   LaserEnd_Ext()
   LIN {X -8.032, Y -15.360, Z 37.400}
   LaserStart_Ext()
   LIN {X 7.075, Y -15.360, Z 37.400}
   LaserEnd_Ext()
   LIN {X 7.240, Y -14.360, Z 37.400}
   LaserStart_Ext()
   LIN {X -7.569, Y -14.360, Z 37.400}
   LaserEnd_Ext()
   LIN {X -7.132, Y -13.360, Z 37.400}
   LaserStart_Ext()
   LIN {X 7.386, Y -13.360, Z 37.400}
   LaserEnd_Ext()
   LIN {X 7.511, Y -12.360, Z 37.400}
   LaserStart_Ext()
   LIN {X -6.697, Y -12.360, Z 37.400}
   LaserEnd_Ext()
   LIN {X -6.262, Y -11.360, Z 37.400}
   LaserStart_Ext()
   LIN {X 7.633, Y -11.360, Z 37.400}
   LaserEnd_Ext()
   LIN {X 7.756, Y -10.360, Z 37.400}
   LaserStart_Ext()
   LIN {X -5.884, Y -10.360, Z 37.400}
   LaserEnd_Ext()
   LIN {X -5.510, Y -9.360, Z 37.400}
   LaserStart_Ext()
   LIN {X 7.878, Y -9.360, Z 37.400}
   LaserEnd_Ext()
   LIN {X 7.959, Y -8.360, Z 37.400}
   LaserStart_Ext()
   LIN {X -5.135, Y -8.360, Z 37.400}
   LaserEnd_Ext()
   LIN {X -4.781, Y -7.360, Z 37.400}
   LaserStart_Ext()
   LIN {X 8.036, Y -7.360, Z 37.400}
   LaserEnd_Ext()
   LIN {X 8.113, Y -6.360, Z 37.400}
   LaserStart_Ext()
   LIN {X -4.476, Y -6.360, Z 37.400}
   LaserEnd_Ext()
   LIN {X -4.171, Y -5.360, Z 37.400}
   LaserStart_Ext()
   LIN {X 8.190, Y -5.360, Z 37.400}
   LaserEnd_Ext()
   LIN {X 8.267, Y -4.360, Z 37.400}
   LaserStart_Ext()
   LIN {X -3.865, Y -4.360, Z 37.400}
   LaserEnd_Ext()
   LIN {X -3.560, Y -3.360, Z 37.400}
   LaserStart_Ext()
   LIN {X 8.311, Y -3.360, Z 37.400}
   LaserEnd_Ext()
   LIN {X 8.326, Y -2.360, Z 37.400}
   LaserStart_Ext()
   LIN {X -3.286, Y -2.360, Z 37.400}
   LaserEnd_Ext()
   LIN {X -3.068, Y -1.360, Z 37.400}
   LaserStart_Ext()
   LIN {X 8.340, Y -1.360, Z 37.400}
   LaserEnd_Ext()
   LIN {X 8.355, Y -0.360, Z 37.400}
   LaserStart_Ext()
   LIN {X -2.851, Y -0.360, Z 37.400}
   LaserEnd_Ext()
   LIN {X -2.634, Y 0.640, Z 37.400}
   LaserStart_Ext()
   LIN {X 8.370, Y 0.640, Z 37.400}
   LaserEnd_Ext()
   LIN {X 8.384, Y 1.640, Z 37.400}
   LaserStart_Ext()
   LIN {X -2.417, Y 1.640, Z 37.400}
   LaserEnd_Ext()
   LIN {X -2.200, Y 2.640, Z 37.400}
   LaserStart_Ext()
   LIN {X 8.399, Y 2.640, Z 37.400}
   LaserEnd_Ext()
   LIN {X 8.413, Y 3.640, Z 37.400}
   LaserStart_Ext()
   LIN {X -1.983, Y 3.640, Z 37.400}
   LaserEnd_Ext()
   LIN {X -1.807, Y 4.640, Z 37.400}
   LaserStart_Ext()
   LIN {X 8.408, Y 4.640, Z 37.400}
   LaserEnd_Ext()
   LIN {X 8.352, Y 5.640, Z 37.400}
   LaserStart_Ext()
   LIN {X -1.698, Y 5.640, Z 37.400}
   LaserEnd_Ext()
   LIN {X -1.589, Y 6.640, Z 37.400}
   LaserStart_Ext()
   LIN {X 8.295, Y 6.640, Z 37.400}
   LaserEnd_Ext()
   LIN {X 8.239, Y 7.640, Z 37.400}
   LaserStart_Ext()
   LIN {X -1.481, Y 7.640, Z 37.400}
   LaserEnd_Ext()
   LIN {X -1.372, Y 8.640, Z 37.400}
   LaserStart_Ext()
   LIN {X 8.183, Y 8.640, Z 37.400}
   LaserEnd_Ext()
   LIN {X 8.135, Y 9.640, Z 37.400}
   LaserStart_Ext()
   LIN {X -1.263, Y 9.640, Z 37.400}
   LaserEnd_Ext()
   LIN {X -1.155, Y 10.640, Z 37.400}
   LaserStart_Ext()
   LIN {X 8.088, Y 10.640, Z 37.400}
   LaserEnd_Ext()
   LIN {X 8.007, Y 11.640, Z 37.400}
   LaserStart_Ext()
   LIN {X -1.046, Y 11.640, Z 37.400}
   LaserEnd_Ext()
   LIN {X -0.951, Y 12.640, Z 37.400}
   LaserStart_Ext()
   LIN {X 7.874, Y 12.640, Z 37.400}
   LaserEnd_Ext()
   LIN {X 7.735, Y 13.640, Z 37.400}
   LaserStart_Ext()
   LIN {X -0.969, Y 13.640, Z 37.400}
   LaserEnd_Ext()
   LIN {X -0.974, Y 14.640, Z 37.400}
   LaserStart_Ext()
   LIN {X 7.596, Y 14.640, Z 37.400}
   LaserEnd_Ext()
   LIN {X 7.457, Y 15.640, Z 37.400}
   LaserStart_Ext()
   LIN {X -0.979, Y 15.640, Z 37.400}
   LaserEnd_Ext()
   LIN {X -0.984, Y 16.640, Z 37.400}
   LaserStart_Ext()
   LIN {X 7.318, Y 16.640, Z 37.400}
   LaserEnd_Ext()
   LIN {X 7.179, Y 17.640, Z 37.400}
   LaserStart_Ext()
   LIN {X -0.990, Y 17.640, Z 37.400}
   LaserEnd_Ext()
   LIN {X -0.995, Y 18.640, Z 37.400}
   LaserStart_Ext()
   LIN {X 7.040, Y 18.640, Z 37.400}
   LaserEnd_Ext()
   LIN {X 6.901, Y 19.640, Z 37.400}
   LaserStart_Ext()
   LIN {X -1.000, Y 19.640, Z 37.400}
   LaserEnd_Ext()
   LIN {X -1.005, Y 20.640, Z 37.400}
   LaserStart_Ext()
   LIN {X 6.762, Y 20.640, Z 37.400}
   LaserEnd_Ext()
   LIN {X 6.617, Y 21.640, Z 37.400}
   LaserStart_Ext()
   LIN {X -1.081, Y 21.640, Z 37.400}
   LaserEnd_Ext()
   LIN {X -1.188, Y 22.640, Z 37.400}
   LaserStart_Ext()
   LIN {X 6.443, Y 22.640, Z 37.400}
   LaserEnd_Ext()
   LIN {X 6.225, Y 23.640, Z 37.400}
   LaserStart_Ext()
   LIN {X -1.295, Y 23.640, Z 37.400}
   LaserEnd_Ext()
   LIN {X -1.401, Y 24.640, Z 37.400}
   LaserStart_Ext()
   LIN {X 6.005, Y 24.640, Z 37.400}
   LaserEnd_Ext()
   LIN {X 5.784, Y 25.640, Z 37.400}
   LaserStart_Ext()
   LIN {X -1.508, Y 25.640, Z 37.400}
   LaserEnd_Ext()
   LIN {X -1.615, Y 26.640, Z 37.400}
   LaserStart_Ext()
   LIN {X 5.562, Y 26.640, Z 37.400}
   LaserEnd_Ext()
   LIN {X 5.340, Y 27.640, Z 37.400}
   LaserStart_Ext()
   LIN {X -1.725, Y 27.640, Z 37.400}
   LaserEnd_Ext()
   LIN {X -1.902, Y 28.640, Z 37.400}
   LaserStart_Ext()
   LIN {X 5.103, Y 28.640, Z 37.400}
   LaserEnd_Ext()
   LIN {X 4.836, Y 29.640, Z 37.400}
   LaserStart_Ext()
   LIN {X -2.078, Y 29.640, Z 37.400}
   LaserEnd_Ext()
   LIN {X -2.254, Y 30.640, Z 37.400}
   LaserStart_Ext()
   LIN {X 4.570, Y 30.640, Z 37.400}
   LaserEnd_Ext()
   LIN {X 4.298, Y 31.640, Z 37.400}
   LaserStart_Ext()
   LIN {X -2.465, Y 31.640, Z 37.400}
   LaserEnd_Ext()
   LIN {X -2.684, Y 32.640, Z 37.400}
   LaserStart_Ext()
   LIN {X 4.013, Y 32.640, Z 37.400}
   LaserEnd_Ext()
   LIN {X 3.709, Y 33.640, Z 37.400}
   LaserStart_Ext()
   LIN {X -2.905, Y 33.640, Z 37.400}
   LaserEnd_Ext()
   LIN {X -3.162, Y 34.640, Z 37.400}
   LaserStart_Ext()
   LIN {X 3.405, Y 34.640, Z 37.400}
   LaserEnd_Ext()
   LIN {X 3.089, Y 35.640, Z 37.400}
   LaserStart_Ext()
   LIN {X -3.420, Y 35.640, Z 37.400}
   LaserEnd_Ext()
   LIN {X -3.695, Y 36.640, Z 37.400}
   LaserStart_Ext()
   LIN {X 2.755, Y 36.640, Z 37.400}
   LaserEnd_Ext()
   LIN {X 2.422, Y 37.640, Z 37.400}
   LaserStart_Ext()
   LIN {X -3.984, Y 37.640, Z 37.400}
   LaserEnd_Ext()
   LIN {X -4.286, Y 38.640, Z 37.400}
   LaserStart_Ext()
   LIN {X 2.068, Y 38.640, Z 37.400}
   LaserEnd_Ext()
   LIN {X 1.708, Y 39.640, Z 37.400}
   LaserStart_Ext()
   LIN {X -4.427, Y 39.640, Z 37.400}
   LaserEnd_Ext()
   LIN {X -4.242, Y 40.640, Z 37.400}
   LaserStart_Ext()
   LIN {X 1.335, Y 40.640, Z 37.400}
   LaserEnd_Ext()
   LIN {X 0.726, Y 41.640, Z 37.400}
   LaserStart_Ext()
   LIN {X -3.673, Y 41.640, Z 37.400}
   LaserEnd_Ext()
   LIN {X -2.190, Y -26.841, Z 38.250}
   LaserStart_Ext()
   LIN {X -2.894, Y -26.717, Z 38.250} C_DIS
   LIN {X -4.205, Y -26.480, Z 38.250} C_DIS
   LIN {X -5.706, Y -25.455, Z 38.250} C_DIS
   LIN {X -5.911, Y -25.316, Z 38.250} C_DIS
   LIN {X -6.024, Y -25.134, Z 38.250} C_DIS
   LIN {X -7.009, Y -23.546, Z 38.250} C_DIS
   LIN {X -7.240, Y -21.756, Z 38.250} C_DIS
   LIN {X -7.277, Y -21.477, Z 38.250} C_DIS
   LIN {X -7.180, Y -21.203, Z 38.250} C_DIS
   LIN {X -6.319, Y -18.904, Z 38.250} C_DIS
   LIN {X -4.889, Y -17.604, Z 38.250} C_DIS
   LIN {X -4.667, Y -17.494, Z 38.250} C_DIS
   LIN {X -2.455, Y -16.842, Z 38.250} C_DIS
   LIN {X -1.080, Y -17.080, Z 38.250} C_DIS
   LIN {X -0.380, Y -17.198, Z 38.250} C_DIS
   LIN {X 0.350, Y -17.699, Z 38.250} C_DIS
   LIN {X 1.370, Y -18.402, Z 38.250} C_DIS
   LIN {X 2.014, Y -19.597, Z 38.250} C_DIS
   LIN {X 2.580, Y -20.639, Z 38.250} C_DIS
   LIN {X 2.596, Y -21.477, Z 38.250} C_DIS
   LIN {X 2.616, Y -22.815, Z 38.250} C_DIS
   LIN {X 2.128, Y -23.823, Z 38.250} C_DIS
   LIN {X 1.558, Y -25.016, Z 38.250} C_DIS
   LIN {X 0.417, Y -25.930, Z 38.250} C_DIS
   LIN {X -0.062, Y -26.310, Z 38.250} C_DIS
   LIN {X -1.069, Y -26.560, Z 38.250} C_DIS
   LIN {X -2.190, Y -26.841, Z 38.250}
   LaserEnd_Ext()
   LIN {X 3.341, Y 37.921, Z 38.250}
   LaserStart_Ext()
   LIN {X 2.785, Y 39.477, Z 38.250} C_DIS
   LIN {X 2.692, Y 39.739, Z 38.250} C_DIS
   LIN {X 2.643, Y 39.872, Z 38.250} C_DIS
   LIN {X 2.172, Y 41.130, Z 38.250} C_DIS
   LIN {X 1.504, Y 42.226, Z 38.250} C_DIS
   LIN {X 1.406, Y 42.387, Z 38.250} C_DIS
   LIN {X 1.194, Y 42.537, Z 38.250} C_DIS
   LIN {X -0.010, Y 43.401, Z 38.250} C_DIS
   LIN {X -1.088, Y 43.602, Z 38.250} C_DIS
   LIN {X -1.727, Y 43.719, Z 38.250} C_DIS
   LIN {X -3.855, Y 42.857, Z 38.250} C_DIS
   LIN {X -4.221, Y 42.712, Z 38.250} C_DIS
   LIN {X -5.222, Y 41.313, Z 38.250} C_DIS
   LIN {X -5.456, Y 40.383, Z 38.250} C_DIS
   LIN {X -5.540, Y 39.979, Z 38.250} C_DIS
   LIN {X -5.479, Y 39.534, Z 38.250} C_DIS
   LIN {X -5.349, Y 38.523, Z 38.250} C_DIS
   LIN {X -5.005, Y 37.398, Z 38.250} C_DIS
   LIN {X -4.937, Y 37.165, Z 38.250} C_DIS
   LIN {X -4.538, Y 35.789, Z 38.250} C_DIS
   LIN {X -4.133, Y 34.236, Z 38.250} C_DIS
   LIN {X -3.941, Y 33.495, Z 38.250} C_DIS
   LIN {X -3.664, Y 32.244, Z 38.250} C_DIS
   LIN {X -3.313, Y 30.668, Z 38.250} C_DIS
   LIN {X -3.137, Y 29.697, Z 38.250} C_DIS
   LIN {X -2.748, Y 27.508, Z 38.250} C_DIS
   LIN {X -2.473, Y 24.936, Z 38.250} C_DIS
   LIN {X -2.281, Y 23.139, Z 38.250} C_DIS
   LIN {X -2.204, Y 22.419, Z 38.250} C_DIS
   LIN {X -2.052, Y 21.233, Z 38.250} C_DIS
   LIN {X -2.015, Y 14.085, Z 38.250} C_DIS
   LIN {X -1.954, Y 12.608, Z 38.250} C_DIS
   LIN {X -2.361, Y 8.770, Z 38.250} C_DIS
   LIN {X -2.840, Y 4.366, Z 38.250} C_DIS
   LIN {X -3.751, Y 0.170, Z 38.250} C_DIS
   LIN {X -4.278, Y -2.326, Z 38.250} C_DIS
   LIN {X -4.552, Y -3.298, Z 38.250} C_DIS
   LIN {X -5.670, Y -6.961, Z 38.250} C_DIS
   LIN {X -6.324, Y -8.783, Z 38.250} C_DIS
   LIN {X -7.101, Y -10.858, Z 38.250} C_DIS
   LIN {X -8.557, Y -14.206, Z 38.250} C_DIS
   LIN {X -8.727, Y -14.604, Z 38.250} C_DIS
   LIN {X -8.883, Y -14.923, Z 38.250} C_DIS
   LIN {X -10.257, Y -17.683, Z 38.250} C_DIS
   LIN {X -11.156, Y -20.493, Z 38.250} C_DIS
   LIN {X -11.223, Y -20.704, Z 38.250} C_DIS
   LIN {X -11.210, Y -20.856, Z 38.250} C_DIS
   LIN {X -10.948, Y -24.404, Z 38.250} C_DIS
   LIN {X -9.577, Y -26.945, Z 38.250} C_DIS
   LIN {X -9.172, Y -27.706, Z 38.250} C_DIS
   LIN {X -8.750, Y -28.051, Z 38.250} C_DIS
   LIN {X -6.764, Y -29.691, Z 38.250} C_DIS
   LIN {X -3.576, Y -30.763, Z 38.250} C_DIS
   LIN {X -0.691, Y -30.694, Z 38.250} C_DIS
   LIN {X 2.555, Y -29.390, Z 38.250} C_DIS
   LIN {X 2.660, Y -29.342, Z 38.250} C_DIS
   LIN {X 2.800, Y -29.194, Z 38.250} C_DIS
   LIN {X 5.321, Y -26.624, Z 38.250} C_DIS
   LIN {X 5.995, Y -25.045, Z 38.250} C_DIS
   LIN {X 6.486, Y -23.872, Z 38.250} C_DIS
   LIN {X 7.011, Y -21.492, Z 38.250} C_DIS
   LIN {X 7.191, Y -20.687, Z 38.250} C_DIS
   LIN {X 7.275, Y -20.265, Z 38.250} C_DIS
   LIN {X 7.752, Y -17.779, Z 38.250} C_DIS
   LIN {X 8.260, Y -14.634, Z 38.250} C_DIS
   LIN {X 8.367, Y -13.948, Z 38.250} C_DIS
   LIN {X 8.494, Y -12.877, Z 38.250} C_DIS
   LIN {X 8.929, Y -9.318, Z 38.250} C_DIS
   LIN {X 9.169, Y -6.195, Z 38.250} C_DIS
   LIN {X 9.342, Y -3.768, Z 38.250} C_DIS
   LIN {X 9.340, Y -2.281, Z 38.250} C_DIS
   LIN {X 9.438, Y 4.467, Z 38.250} C_DIS
   LIN {X 9.114, Y 10.228, Z 38.250} C_DIS
   LIN {X 9.077, Y 11.017, Z 38.250} C_DIS
   LIN {X 9.049, Y 11.279, Z 38.250} C_DIS
   LIN {X 7.525, Y 22.243, Z 38.250} C_DIS
   LIN {X 7.508, Y 22.354, Z 38.250} C_DIS
   LIN {X 7.470, Y 22.528, Z 38.250} C_DIS
   LIN {X 6.118, Y 28.626, Z 38.250} C_DIS
   LIN {X 5.689, Y 30.237, Z 38.250} C_DIS
   LIN {X 5.004, Y 32.718, Z 38.250} C_DIS
   LIN {X 4.487, Y 34.418, Z 38.250} C_DIS
   LIN {X 3.908, Y 36.237, Z 38.250} C_DIS
   LIN {X 3.512, Y 37.422, Z 38.250} C_DIS
   LIN {X 3.341, Y 37.921, Z 38.250}
   LaserEnd_Ext()
   LIN {X 7.602, Y -11.930, Z 38.250}
   LaserStart_Ext()
   LIN {X 7.602, Y 14.428, Z 38.250}
   LaserEnd_Ext()
   LIN {X 6.602, Y 21.619, Z 38.250}
   LaserStart_Ext()
   LIN {X 6.602, Y -18.465, Z 38.250}
   LaserEnd_Ext()
   LIN {X 5.602, Y -23.239, Z 38.250}
   LaserStart_Ext()
   LIN {X 5.602, Y 26.334, Z 38.250}
   LaserEnd_Ext()
   LIN {X 4.602, Y 30.417, Z 38.250}
   LaserStart_Ext()
   LIN {X 4.602, Y -25.762, Z 38.250}
   LaserEnd_Ext()
   LIN {X 3.602, Y -26.949, Z 38.250}
   LaserStart_Ext()
   LIN {X 3.602, Y -22.979, Z 38.250}
   LaserEnd_Ext()
   LIN {X 3.602, Y -21.866, Z 38.250}
   LaserStart_Ext()
   LIN {X 3.602, Y 33.891, Z 38.250}
   LaserEnd_Ext()
   LIN {X 2.602, Y 36.989, Z 38.250}
   LaserStart_Ext()
   LIN {X 2.602, Y -18.581, Z 38.250}
   LaserEnd_Ext()
   LIN {X 2.602, Y -25.150, Z 38.250}
   LaserStart_Ext()
   LIN {X 2.602, Y -27.968, Z 38.250}
   LaserEnd_Ext()
   LIN {X 1.602, Y -28.696, Z 38.250}
   LaserStart_Ext()
   LIN {X 1.602, Y -26.262, Z 38.250}
   LaserEnd_Ext()
   LIN {X 1.602, Y -17.348, Z 38.250}
   LaserStart_Ext()
   LIN {X 1.602, Y 39.800, Z 38.250}
   LaserEnd_Ext()
   LIN {X 0.602, Y 41.732, Z 38.250}
   LaserStart_Ext()
   LIN {X 0.602, Y -16.659, Z 38.250}
   LaserEnd_Ext()
   LIN {X 0.602, Y -27.060, Z 38.250}
   LaserStart_Ext()
   LIN {X 0.602, Y -29.097, Z 38.250}
   LaserEnd_Ext()
   LIN {X -0.398, Y -29.499, Z 38.250}
   LaserStart_Ext()
   LIN {X -0.398, Y -27.424, Z 38.250}
   LaserEnd_Ext()
   LIN {X -0.398, Y -16.181, Z 38.250}
   LaserStart_Ext()
   LIN {X -0.398, Y 42.449, Z 38.250}
   LaserEnd_Ext()
   LIN {X -1.398, Y 42.642, Z 38.250}
   LaserStart_Ext()
   LIN {X -1.398, Y 24.288, Z 38.250}
   LaserEnd_Ext()
   LIN {X -1.398, Y 8.374, Z 38.250}
   LaserStart_Ext()
   LIN {X -1.398, Y -16.010, Z 38.250}
   LaserEnd_Ext()
   LIN {X -1.398, Y -27.674, Z 38.250}
   LaserStart_Ext()
   LIN {X -1.398, Y -29.713, Z 38.250}
   LaserEnd_Ext()
   LIN {X -2.398, Y -29.741, Z 38.250}
   LaserStart_Ext()
   LIN {X -2.398, Y -27.820, Z 38.250}
   LaserEnd_Ext()
   LIN {X -2.398, Y -15.845, Z 38.250}
   LaserStart_Ext()
   LIN {X -2.398, Y 1.687, Z 38.250}
   LaserEnd_Ext()
   LIN {X -2.398, Y 31.160, Z 38.250}
   LaserStart_Ext()
   LIN {X -2.398, Y 42.369, Z 38.250}
   LaserEnd_Ext()
   LIN {X -3.398, Y 41.964, Z 38.250}
   LaserStart_Ext()
   LIN {X -3.398, Y 35.380, Z 38.250}
   LaserEnd_Ext()
   LIN {X -3.398, Y -2.891, Z 38.250}
   LaserStart_Ext()
   LIN {X -3.398, Y -16.078, Z 38.250}
   LaserEnd_Ext()
   LIN {X -3.398, Y -27.642, Z 38.250}
   LaserStart_Ext()
   LIN {X -3.398, Y -29.768, Z 38.250}
   LaserEnd_Ext()
   LIN {X -4.398, Y -29.432, Z 38.250}
   LaserStart_Ext()
   LIN {X -4.398, Y -27.460, Z 38.250}
   LaserEnd_Ext()
   LIN {X -4.398, Y -16.372, Z 38.250}
   LaserStart_Ext()
   LIN {X -4.398, Y -6.218, Z 38.250}
   LaserEnd_Ext()
   LIN {X -4.398, Y 38.969, Z 38.250}
   LaserStart_Ext()
   LIN {X -4.398, Y 40.489, Z 38.250}
   LaserEnd_Ext()
   LIN {X -5.398, Y -9.162, Z 38.250}
   LaserStart_Ext()
   LIN {X -5.398, Y -16.724, Z 38.250}
   LaserEnd_Ext()
   LIN {X -5.398, Y -26.876, Z 38.250}
   LaserStart_Ext()
   LIN {X -5.398, Y -29.096, Z 38.250}
   LaserEnd_Ext()
   LIN {X -6.398, Y -28.696, Z 38.250}
   LaserStart_Ext()
   LIN {X -6.398, Y -26.194, Z 38.250}
   LaserEnd_Ext()
   LIN {X -6.398, Y -17.624, Z 38.250}
   LaserStart_Ext()
   LIN {X -6.398, Y -11.749, Z 38.250}
   LaserEnd_Ext()
   LIN {X -7.398, Y -14.049, Z 38.250}
   LaserStart_Ext()
   LIN {X -7.398, Y -18.934, Z 38.250}
   LaserEnd_Ext()
   LIN {X -7.398, Y -24.816, Z 38.250}
   LaserStart_Ext()
   LIN {X -7.398, Y -27.871, Z 38.250}
   LaserEnd_Ext()
   LIN {X -8.398, Y -27.033, Z 38.250}
   LaserStart_Ext()
   LIN {X -8.398, Y -16.192, Z 38.250}
   LaserEnd_Ext()
   LIN {X -9.398, Y -18.279, Z 38.250}
   LaserStart_Ext()
   LIN {X -9.398, Y -25.170, Z 38.250}
   LaserEnd_Ext()
   LIN {X -0.315, Y -17.145, Z 39.100}
   LaserStart_Ext()
   LIN {X 1.149, Y -18.149, Z 39.100} C_DIS
   LIN {X 1.438, Y -18.345, Z 39.100} C_DIS
   LIN {X 1.638, Y -18.710, Z 39.100} C_DIS
   LIN {X 2.654, Y -20.579, Z 39.100} C_DIS
   LIN {X 2.694, Y -22.707, Z 39.100} C_DIS
   LIN {X 1.640, Y -24.960, Z 39.100} C_DIS
   LIN {X 0.780, Y -25.649, Z 39.100} C_DIS
   LIN {X 0.024, Y -26.257, Z 39.100} C_DIS
   LIN {X -0.590, Y -26.413, Z 39.100} C_DIS
   LIN {X -2.102, Y -26.792, Z 39.100} C_DIS
   LIN {X -4.039, Y -26.450, Z 39.100} C_DIS
   LIN {X -4.208, Y -26.374, Z 39.100} C_DIS
   LIN {X -5.827, Y -25.276, Z 39.100} C_DIS
   LIN {X -6.722, Y -23.842, Z 39.100} C_DIS
   LIN {X -6.929, Y -23.508, Z 39.100} C_DIS
   LIN {X -6.977, Y -23.132, Z 39.100} C_DIS
   LIN {X -7.201, Y -21.440, Z 39.100} C_DIS
   LIN {X -6.612, Y -19.780, Z 39.100} C_DIS
   LIN {X -6.291, Y -18.921, Z 39.100} C_DIS
   LIN {X -5.757, Y -18.435, Z 39.100} C_DIS
   LIN {X -4.756, Y -17.498, Z 39.100} C_DIS
   LIN {X -2.486, Y -16.822, Z 39.100} C_DIS
   LIN {X -2.334, Y -16.804, Z 39.100} C_DIS
   LIN {X -0.315, Y -17.145, Z 39.100}
   LaserEnd_Ext()
   LIN {X 4.937, Y 32.834, Z 39.100}
   LaserStart_Ext()
   LIN {X 4.702, Y 33.610, Z 39.100} C_DIS
   LIN {X 3.734, Y 36.647, Z 39.100} C_DIS
   LIN {X 3.284, Y 37.964, Z 39.100} C_DIS
   LIN {X 3.129, Y 38.396, Z 39.100} C_DIS
   LIN {X 2.636, Y 39.768, Z 39.100} C_DIS
   LIN {X 2.116, Y 41.148, Z 39.100} C_DIS
   LIN {X 1.332, Y 42.444, Z 39.100} C_DIS
   LIN {X 0.139, Y 43.295, Z 39.100} C_DIS
   LIN {X -0.086, Y 43.454, Z 39.100} C_DIS
   LIN {X -0.617, Y 43.551, Z 39.100} C_DIS
   LIN {X -1.804, Y 43.769, Z 39.100} C_DIS
   LIN {X -2.601, Y 43.446, Z 39.100} C_DIS
   LIN {X -4.278, Y 42.771, Z 39.100} C_DIS
   LIN {X -5.066, Y 41.635, Z 39.100} C_DIS
   LIN {X -5.348, Y 41.235, Z 39.100} C_DIS
   LIN {X -5.411, Y 40.939, Z 39.100} C_DIS
   LIN {X -5.610, Y 39.982, Z 39.100} C_DIS
   LIN {X -5.450, Y 38.813, Z 39.100} C_DIS
   LIN {X -5.414, Y 38.564, Z 39.100} C_DIS
   LIN {X -5.356, Y 38.377, Z 39.100} C_DIS
   LIN {X -5.046, Y 37.368, Z 39.100} C_DIS
   LIN {X -4.693, Y 36.162, Z 39.100} C_DIS
   LIN {X -4.597, Y 35.833, Z 39.100} C_DIS
   LIN {X -4.434, Y 35.207, Z 39.100} C_DIS
   LIN {X -3.994, Y 33.539, Z 39.100} C_DIS
   LIN {X -3.673, Y 32.120, Z 39.100} C_DIS
   LIN {X -3.359, Y 30.714, Z 39.100} C_DIS
   LIN {X -2.838, Y 27.832, Z 39.100} C_DIS
   LIN {X -2.787, Y 27.556, Z 39.100} C_DIS
   LIN {X -2.482, Y 24.705, Z 39.100} C_DIS
   LIN {X -2.353, Y 23.493, Z 39.100} C_DIS
   LIN {X -2.097, Y 21.497, Z 39.100} C_DIS
   LIN {X -2.064, Y 15.178, Z 39.100} C_DIS
   LIN {X -1.959, Y 12.611, Z 39.100} C_DIS
   LIN {X -2.666, Y 5.940, Z 39.100} C_DIS
   LIN {X -2.843, Y 4.309, Z 39.100} C_DIS
   LIN {X -3.180, Y 2.756, Z 39.100} C_DIS
   LIN {X -4.227, Y -2.202, Z 39.100} C_DIS
   LIN {X -4.772, Y -4.132, Z 39.100} C_DIS
   LIN {X -5.541, Y -6.652, Z 39.100} C_DIS
   LIN {X -6.740, Y -9.994, Z 39.100} C_DIS
   LIN {X -7.039, Y -10.793, Z 39.100} C_DIS
   LIN {X -7.599, Y -12.080, Z 39.100} C_DIS
   LIN {X -8.627, Y -14.480, Z 39.100} C_DIS
   LIN {X -9.566, Y -16.399, Z 39.100} C_DIS
   LIN {X -10.191, Y -17.653, Z 39.100} C_DIS
   LIN {X -10.599, Y -18.930, Z 39.100} C_DIS
   LIN {X -11.149, Y -20.676, Z 39.100} C_DIS
   LIN {X -11.046, Y -21.940, Z 39.100} C_DIS
   LIN {X -10.865, Y -24.376, Z 39.100} C_DIS
   LIN {X -9.367, Y -27.154, Z 39.100} C_DIS
   LIN {X -9.082, Y -27.674, Z 39.100} C_DIS
   LIN {X -8.700, Y -27.993, Z 39.100} C_DIS
   LIN {X -6.732, Y -29.617, Z 39.100} C_DIS
   LIN {X -4.570, Y -30.344, Z 39.100} C_DIS
   LIN {X -3.417, Y -30.730, Z 39.100} C_DIS
   LIN {X -2.188, Y -30.662, Z 39.100} C_DIS
   LIN {X -0.453, Y -30.614, Z 39.100} C_DIS
   LIN {X 1.494, Y -29.832, Z 39.100} C_DIS
   LIN {X 2.883, Y -29.187, Z 39.100} C_DIS
   LIN {X 4.742, Y -27.235, Z 39.100} C_DIS
   LIN {X 5.413, Y -26.552, Z 39.100} C_DIS
   LIN {X 5.592, Y -26.132, Z 39.100} C_DIS
   LIN {X 6.568, Y -23.803, Z 39.100} C_DIS
   LIN {X 7.099, Y -21.392, Z 39.100} C_DIS
   LIN {X 7.265, Y -20.616, Z 39.100} C_DIS
   LIN {X 7.478, Y -19.484, Z 39.100} C_DIS
   LIN {X 7.819, Y -17.707, Z 39.100} C_DIS
   LIN {X 8.077, Y -16.110, Z 39.100} C_DIS
   LIN {X 8.423, Y -13.892, Z 39.100} C_DIS
   LIN {X 8.831, Y -10.433, Z 39.100} C_DIS
   LIN {X 8.974, Y -9.261, Z 39.100} C_DIS
   LIN {X 9.053, Y -8.233, Z 39.100} C_DIS
   LIN {X 9.376, Y -3.680, Z 39.100} C_DIS
   LIN {X 9.374, Y -0.891, Z 39.100} C_DIS
   LIN {X 9.453, Y 4.552, Z 39.100} C_DIS
   LIN {X 9.129, Y 10.300, Z 39.100} C_DIS
   LIN {X 9.051, Y 11.219, Z 39.100} C_DIS
   LIN {X 8.866, Y 12.442, Z 39.100} C_DIS
   LIN {X 7.477, Y 22.438, Z 39.100} C_DIS
   LIN {X 6.434, Y 27.075, Z 39.100} C_DIS
   LIN {X 6.067, Y 28.732, Z 39.100} C_DIS
   LIN {X 5.962, Y 29.123, Z 39.100} C_DIS
   LIN {X 4.937, Y 32.834, Z 39.100}
   LaserEnd_Ext()
   LIN {X -0.546, Y 42.522, Z 39.100}
   LaserStart_Ext()
   LIN {X -2.219, Y 42.522, Z 39.100}
   LaserEnd_Ext()
   LIN {X -3.928, Y 41.522, Z 39.100}
   LaserStart_Ext()
   LIN {X 0.724, Y 41.522, Z 39.100}
   LaserEnd_Ext()
   LIN {X 1.283, Y 40.522, Z 39.100}
   LaserStart_Ext()
   LIN {X -4.476, Y 40.522, Z 39.100}
   LaserEnd_Ext()
   LIN {X -4.538, Y 39.522, Z 39.100}
   LaserStart_Ext()
   LIN {X 1.660, Y 39.522, Z 39.100}
   LaserEnd_Ext()
   LIN {X 2.021, Y 38.522, Z 39.100}
   LaserStart_Ext()
   LIN {X -4.354, Y 38.522, Z 39.100}
   LaserEnd_Ext()
   LIN {X -4.049, Y 37.522, Z 39.100}
   LaserStart_Ext()
   LIN {X 2.378, Y 37.522, Z 39.100}
   LaserEnd_Ext()
   LIN {X 2.721, Y 36.522, Z 39.100}
   LaserStart_Ext()
   LIN {X -3.756, Y 36.522, Z 39.100}
   LaserEnd_Ext()
   LIN {X -3.482, Y 35.522, Z 39.100}
   LaserStart_Ext()
   LIN {X 3.043, Y 35.522, Z 39.100}
   LaserEnd_Ext()
   LIN {X 3.362, Y 34.522, Z 39.100}
   LaserStart_Ext()
   LIN {X -3.219, Y 34.522, Z 39.100}
   LaserEnd_Ext()
   LIN {X -2.965, Y 33.522, Z 39.100}
   LaserStart_Ext()
   LIN {X 3.680, Y 33.522, Z 39.100}
   LaserEnd_Ext()
   LIN {X 3.986, Y 32.522, Z 39.100}
   LaserStart_Ext()
   LIN {X -2.739, Y 32.522, Z 39.100}
   LaserEnd_Ext()
   LIN {X -2.515, Y 31.522, Z 39.100}
   LaserStart_Ext()
   LIN {X 4.262, Y 31.522, Z 39.100}
   LaserEnd_Ext()
   LIN {X 4.539, Y 30.522, Z 39.100}
   LaserStart_Ext()
   LIN {X -2.308, Y 30.522, Z 39.100}
   LaserEnd_Ext()
   LIN {X -2.127, Y 29.522, Z 39.100}
   LaserStart_Ext()
   LIN {X 4.815, Y 29.522, Z 39.100}
   LaserEnd_Ext()
   LIN {X 5.088, Y 28.522, Z 39.100}
   LaserStart_Ext()
   LIN {X -1.946, Y 28.522, Z 39.100}
   LaserEnd_Ext()
   LIN {X -1.778, Y 27.522, Z 39.100}
   LaserStart_Ext()
   LIN {X 5.311, Y 27.522, Z 39.100}
   LaserEnd_Ext()
   LIN {X 5.534, Y 26.522, Z 39.100}
   LaserStart_Ext()
   LIN {X -1.671, Y 26.522, Z 39.100}
   LaserEnd_Ext()
   LIN {X -1.564, Y 25.522, Z 39.100}
   LaserStart_Ext()
   LIN {X 5.759, Y 25.522, Z 39.100}
   LaserEnd_Ext()
   LIN {X 5.984, Y 24.522, Z 39.100}
   LaserStart_Ext()
   LIN {X -1.457, Y 24.522, Z 39.100}
   LaserEnd_Ext()
   LIN {X -1.348, Y 23.522, Z 39.100}
   LaserStart_Ext()
   LIN {X 6.209, Y 23.522, Z 39.100}
   LaserEnd_Ext()
   LIN {X 6.434, Y 22.522, Z 39.100}
   LaserStart_Ext()
   LIN {X -1.220, Y 22.522, Z 39.100}
   LaserEnd_Ext()
   LIN {X -1.099, Y 21.522, Z 39.100}
   LaserStart_Ext()
   LIN {X 6.595, Y 21.522, Z 39.100}
   LaserEnd_Ext()
   LIN {X 6.734, Y 20.522, Z 39.100}
   LaserStart_Ext()
   LIN {X -1.092, Y 20.522, Z 39.100}
   LaserEnd_Ext()
   LIN {X -1.087, Y 19.522, Z 39.100}
   LaserStart_Ext()
   LIN {X 6.873, Y 19.522, Z 39.100}
   LaserEnd_Ext()
   LIN {X 7.012, Y 18.522, Z 39.100}
   LaserStart_Ext()
   LIN {X -1.082, Y 18.522, Z 39.100}
   LaserEnd_Ext()
   LIN {X -1.076, Y 17.522, Z 39.100}
   LaserStart_Ext()
   LIN {X 7.151, Y 17.522, Z 39.100}
   LaserEnd_Ext()
   LIN {X 7.290, Y 16.522, Z 39.100}
   LaserStart_Ext()
   LIN {X -1.071, Y 16.522, Z 39.100}
   LaserEnd_Ext()
   LIN {X -1.066, Y 15.522, Z 39.100}
   LaserStart_Ext()
   LIN {X 7.429, Y 15.522, Z 39.100}
   LaserEnd_Ext()
   LIN {X 7.568, Y 14.522, Z 39.100}
   LaserStart_Ext()
   LIN {X -1.037, Y 14.522, Z 39.100}
   LaserEnd_Ext()
   LIN {X -0.996, Y 13.522, Z 39.100}
   LaserStart_Ext()
   LIN {X 7.707, Y 13.522, Z 39.100}
   LaserEnd_Ext()
   LIN {X 7.846, Y 12.522, Z 39.100}
   LaserStart_Ext()
   LIN {X -0.964, Y 12.522, Z 39.100}
   LaserEnd_Ext()
   LIN {X -1.069, Y 11.522, Z 39.100}
   LaserStart_Ext()
   LIN {X 7.994, Y 11.522, Z 39.100}
   LaserEnd_Ext()
   LIN {X 8.107, Y 10.522, Z 39.100}
   LaserStart_Ext()
   LIN {X -1.175, Y 10.522, Z 39.100}
   LaserEnd_Ext()
   LIN {X -1.281, Y 9.522, Z 39.100}
   LaserStart_Ext()
   LIN {X 8.171, Y 9.522, Z 39.100}
   LaserEnd_Ext()
   LIN {X 8.228, Y 8.522, Z 39.100}
   LaserStart_Ext()
   LIN {X -1.387, Y 8.522, Z 39.100}
   LaserEnd_Ext()
   LIN {X -1.493, Y 7.522, Z 39.100}
   LaserStart_Ext()
   LIN {X 8.284, Y 7.522, Z 39.100}
   LaserEnd_Ext()
   LIN {X 8.340, Y 6.522, Z 39.100}
   LaserStart_Ext()
   LIN {X -1.599, Y 6.522, Z 39.100}
   LaserEnd_Ext()
   LIN {X -1.705, Y 5.522, Z 39.100}
   LaserStart_Ext()
   LIN {X 8.396, Y 5.522, Z 39.100}
   LaserEnd_Ext()
   LIN {X 8.452, Y 4.522, Z 39.100}
   LaserStart_Ext()
   LIN {X -1.814, Y 4.522, Z 39.100}
   LaserEnd_Ext()
   LIN {X -1.991, Y 3.522, Z 39.100}
   LaserStart_Ext()
   LIN {X 8.438, Y 3.522, Z 39.100}
   LaserEnd_Ext()
   LIN {X 8.423, Y 2.522, Z 39.100}
   LaserStart_Ext()
   LIN {X -2.208, Y 2.522, Z 39.100}
   LaserEnd_Ext()
   LIN {X -2.419, Y 1.522, Z 39.100}
   LaserStart_Ext()
   LIN {X 8.409, Y 1.522, Z 39.100}
   LaserEnd_Ext()
   LIN {X 8.394, Y 0.522, Z 39.100}
   LaserStart_Ext()
   LIN {X -2.630, Y 0.522, Z 39.100}
   LaserEnd_Ext()
   LIN {X -2.841, Y -0.478, Z 39.100}
   LaserStart_Ext()
   LIN {X 8.379, Y -0.478, Z 39.100}
   LaserEnd_Ext()
   LIN {X 8.374, Y -1.478, Z 39.100}
   LaserStart_Ext()
   LIN {X -3.052, Y -1.478, Z 39.100}
   LaserEnd_Ext()
   LIN {X -3.266, Y -2.478, Z 39.100}
   LaserStart_Ext()
   LIN {X 8.375, Y -2.478, Z 39.100}
   LaserEnd_Ext()
   LIN {X 8.376, Y -3.478, Z 39.100}
   LaserStart_Ext()
   LIN {X -3.548, Y -3.478, Z 39.100}
   LaserEnd_Ext()
   LIN {X -3.832, Y -4.478, Z 39.100}
   LaserStart_Ext()
   LIN {X 8.317, Y -4.478, Z 39.100}
   LaserEnd_Ext()
   LIN {X 8.246, Y -5.478, Z 39.100}
   LaserStart_Ext()
   LIN {X -4.137, Y -5.478, Z 39.100}
   LaserEnd_Ext()
   LIN {X -4.443, Y -6.478, Z 39.100}
   LaserStart_Ext()
   LIN {X 8.175, Y -6.478, Z 39.100}
   LaserEnd_Ext()
   LIN {X 8.104, Y -7.478, Z 39.100}
   LaserStart_Ext()
   LIN {X -4.775, Y -7.478, Z 39.100}
   LaserEnd_Ext()
   LIN {X -5.134, Y -8.478, Z 39.100}
   LaserStart_Ext()
   LIN {X 8.031, Y -8.478, Z 39.100}
   LaserEnd_Ext()
   LIN {X 7.940, Y -9.478, Z 39.100}
   LaserStart_Ext()
   LIN {X -5.493, Y -9.478, Z 39.100}
   LaserEnd_Ext()
   LIN {X -5.854, Y -10.478, Z 39.100}
   LaserStart_Ext()
   LIN {X 7.818, Y -10.478, Z 39.100}
   LaserEnd_Ext()
   LIN {X 7.700, Y -11.478, Z 39.100}
   LaserStart_Ext()
   LIN {X -6.247, Y -11.478, Z 39.100}
   LaserEnd_Ext()
   LIN {X -6.682, Y -12.478, Z 39.100}
   LaserStart_Ext()
   LIN {X 7.583, Y -12.478, Z 39.100}
   LaserEnd_Ext()
   LIN {X 7.465, Y -13.478, Z 39.100}
   LaserStart_Ext()
   LIN {X -7.110, Y -13.478, Z 39.100}
   LaserEnd_Ext()
   LIN {X -7.538, Y -14.478, Z 39.100}
   LaserStart_Ext()
   LIN {X 7.319, Y -14.478, Z 39.100}
   LaserEnd_Ext()
   LIN {X 7.163, Y -15.478, Z 39.100}
   LaserStart_Ext()
   LIN {X -8.002, Y -15.478, Z 39.100}
   LaserEnd_Ext()
   LIN {X -8.492, Y -16.478, Z 39.100}
   LaserStart_Ext()
   LIN {X -4.836, Y -16.478, Z 39.100}
   LaserEnd_Ext()
   LIN {X 0.481, Y -16.478, Z 39.100}
   LaserStart_Ext()
   LIN {X 7.004, Y -16.478, Z 39.100}
   LaserEnd_Ext()
   LIN {X 6.843, Y -17.478, Z 39.100}
   LaserStart_Ext()
   LIN {X 1.942, Y -17.478, Z 39.100}
   LaserEnd_Ext()
   LIN {X -6.198, Y -17.478, Z 39.100}
   LaserStart_Ext()
   LIN {X -8.987, Y -17.478, Z 39.100}
   LaserEnd_Ext()
   LIN {X -9.405, Y -18.478, Z 39.100}
   LaserStart_Ext()
   LIN {X -7.187, Y -18.478, Z 39.100}
   LaserEnd_Ext()
   LIN {X 2.650, Y -18.478, Z 39.100}
   LaserStart_Ext()
   LIN {X 6.652, Y -18.478, Z 39.100}
   LaserEnd_Ext()
   LIN {X 6.461, Y -19.478, Z 39.100}
   LaserStart_Ext()
   LIN {X 3.194, Y -19.478, Z 39.100}
   LaserEnd_Ext()
   LIN {X -7.567, Y -19.478, Z 39.100}
   LaserStart_Ext()
   LIN {X -9.724, Y -19.478, Z 39.100}
   LaserEnd_Ext()
   LIN {X -10.038, Y -20.478, Z 39.100}
   LaserStart_Ext()
   LIN {X -7.921, Y -20.478, Z 39.100}
   LaserEnd_Ext()
   LIN {X 3.648, Y -20.478, Z 39.100}
   LaserStart_Ext()
   LIN {X 6.272, Y -20.478, Z 39.100}
   LaserEnd_Ext()
   LIN {X 6.056, Y -21.478, Z 39.100}
   LaserStart_Ext()
   LIN {X 3.671, Y -21.478, Z 39.100}
   LaserEnd_Ext()
   LIN {X -8.201, Y -21.478, Z 39.100}
   LaserStart_Ext()
   LIN {X -10.080, Y -21.478, Z 39.100}
   LaserEnd_Ext()
   LIN {X -10.003, Y -22.478, Z 39.100}
   LaserStart_Ext()
   LIN {X -8.073, Y -22.478, Z 39.100}
   LaserEnd_Ext()
   LIN {X 3.690, Y -22.478, Z 39.100}
   LaserStart_Ext()
   LIN {X 5.836, Y -22.478, Z 39.100}
   LaserEnd_Ext()
   LIN {X 5.615, Y -23.478, Z 39.100}
   LaserStart_Ext()
   LIN {X 3.457, Y -23.478, Z 39.100}
   LaserEnd_Ext()
   LIN {X -7.941, Y -23.478, Z 39.100}
   LaserStart_Ext()
   LIN {X -9.929, Y -23.478, Z 39.100}
   LaserEnd_Ext()
   LIN {X -9.674, Y -24.478, Z 39.100}
   LaserStart_Ext()
   LIN {X -7.504, Y -24.478, Z 39.100}
   LaserEnd_Ext()
   LIN {X 2.979, Y -24.478, Z 39.100}
   LaserStart_Ext()
   LIN {X 5.201, Y -24.478, Z 39.100}
   LaserEnd_Ext()
   LIN {X 4.782, Y -25.478, Z 39.100}
   LaserStart_Ext()
   LIN {X 2.495, Y -25.478, Z 39.100}
   LaserEnd_Ext()
   LIN {X -6.879, Y -25.478, Z 39.100}
   LaserStart_Ext()
   LIN {X -9.134, Y -25.478, Z 39.100}
   LaserEnd_Ext()
   LIN {X -8.595, Y -26.478, Z 39.100}
   LaserStart_Ext()
   LIN {X -5.835, Y -26.478, Z 39.100}
   LaserEnd_Ext()
   LIN {X 1.344, Y -26.478, Z 39.100}
   LaserStart_Ext()
   LIN {X 4.084, Y -26.478, Z 39.100}
   LaserEnd_Ext()
   LIN {X 3.130, Y -27.478, Z 39.100}
   LaserStart_Ext()
   LIN {X -0.726, Y -27.478, Z 39.100}
   LaserEnd_Ext()
   LIN {X -3.966, Y -27.478, Z 39.100}
   LaserStart_Ext()
   LIN {X -7.752, Y -27.478, Z 39.100}
   LaserEnd_Ext()
   LIN {X -6.541, Y -28.478, Z 39.100}
   LaserStart_Ext()
   LIN {X 2.035, Y -28.478, Z 39.100}
   LaserEnd_Ext()
   LIN {X -0.308, Y -29.478, Z 39.100}
   LaserStart_Ext()
   LIN {X -4.007, Y -29.478, Z 39.100}
   LaserEnd_Ext()
   LIN {X -4.691, Y -17.456, Z 39.950}
   LaserStart_Ext()
   LIN {X -3.638, Y -17.142, Z 39.950} C_DIS
   LIN {X -2.328, Y -16.746, Z 39.950} C_DIS
   LIN {X -0.755, Y -17.006, Z 39.950} C_DIS
   LIN {X -0.250, Y -17.092, Z 39.950} C_DIS
   LIN {X 0.094, Y -17.327, Z 39.950} C_DIS
   LIN {X 1.506, Y -18.288, Z 39.950} C_DIS
   LIN {X 2.484, Y -20.071, Z 39.950} C_DIS
   LIN {X 2.728, Y -20.518, Z 39.950} C_DIS
   LIN {X 2.738, Y -21.055, Z 39.950} C_DIS
   LIN {X 2.773, Y -22.694, Z 39.950} C_DIS
   LIN {X 1.923, Y -24.477, Z 39.950} C_DIS
   LIN {X 1.732, Y -24.892, Z 39.950} C_DIS
   LIN {X 1.292, Y -25.253, Z 39.950} C_DIS
   LIN {X 0.111, Y -26.203, Z 39.950} C_DIS
   LIN {X -1.760, Y -26.680, Z 39.950} C_DIS
   LIN {X -2.014, Y -26.743, Z 39.950} C_DIS
   LIN {X -2.372, Y -26.680, Z 39.950} C_DIS
   LIN {X -4.030, Y -26.391, Z 39.950} C_DIS
   LIN {X -5.098, Y -25.672, Z 39.950} C_DIS
   LIN {X -5.742, Y -25.235, Z 39.950} C_DIS
   LIN {X -6.222, Y -24.467, Z 39.950} C_DIS
   LIN {X -6.848, Y -23.471, Z 39.950} C_DIS
   LIN {X -7.013, Y -22.255, Z 39.950} C_DIS
   LIN {X -7.126, Y -21.403, Z 39.950} C_DIS
   LIN {X -6.632, Y -20.009, Z 39.950} C_DIS
   LIN {X -6.232, Y -18.895, Z 39.950} C_DIS
   LIN {X -5.712, Y -18.412, Z 39.950} C_DIS
   LIN {X -4.691, Y -17.456, Z 39.950}
   LaserEnd_Ext()
   LIN {X -2.142, Y 21.760, Z 39.950}
   LaserStart_Ext()
   LIN {X -2.502, Y 24.567, Z 39.950} C_DIS
   LIN {X -2.684, Y 26.271, Z 39.950} C_DIS
   LIN {X -2.826, Y 27.603, Z 39.950} C_DIS
   LIN {X -3.244, Y 29.885, Z 39.950} C_DIS
   LIN {X -3.406, Y 30.760, Z 39.950} C_DIS
   LIN {X -3.696, Y 32.032, Z 39.950} C_DIS
   LIN {X -4.047, Y 33.584, Z 39.950} C_DIS
   LIN {X -4.261, Y 34.395, Z 39.950} C_DIS
   LIN {X -4.655, Y 35.875, Z 39.950} C_DIS
   LIN {X -5.094, Y 37.364, Z 39.950} C_DIS
   LIN {X -5.479, Y 38.605, Z 39.950} C_DIS
   LIN {X -5.650, Y 39.786, Z 39.950} C_DIS
   LIN {X -5.679, Y 39.997, Z 39.950} C_DIS
   LIN {X -5.622, Y 40.258, Z 39.950} C_DIS
   LIN {X -5.396, Y 41.334, Z 39.950} C_DIS
   LIN {X -4.720, Y 42.292, Z 39.950} C_DIS
   LIN {X -4.330, Y 42.836, Z 39.950} C_DIS
   LIN {X -3.909, Y 43.003, Z 39.950} C_DIS
   LIN {X -1.882, Y 43.818, Z 39.950} C_DIS
   LIN {X -1.118, Y 43.682, Z 39.950} C_DIS
   LIN {X -0.163, Y 43.508, Z 39.950} C_DIS
   LIN {X 1.235, Y 42.516, Z 39.950} C_DIS
   LIN {X 2.030, Y 41.247, Z 39.950} C_DIS
   LIN {X 2.488, Y 40.039, Z 39.950} C_DIS
   LIN {X 2.581, Y 39.792, Z 39.950} C_DIS
   LIN {X 2.731, Y 39.377, Z 39.950} C_DIS
   LIN {X 3.267, Y 37.893, Z 39.950} C_DIS
   LIN {X 3.554, Y 37.055, Z 39.950} C_DIS
   LIN {X 3.936, Y 35.912, Z 39.950} C_DIS
   LIN {X 4.856, Y 32.997, Z 39.950} C_DIS
   LIN {X 4.920, Y 32.781, Z 39.950} C_DIS
   LIN {X 6.015, Y 28.838, Z 39.950} C_DIS
   LIN {X 6.322, Y 27.525, Z 39.950} C_DIS
   LIN {X 7.442, Y 22.548, Z 39.950} C_DIS
   LIN {X 8.442, Y 15.351, Z 39.950} C_DIS
   LIN {X 8.989, Y 11.729, Z 39.950} C_DIS
   LIN {X 9.221, Y 9.006, Z 39.950} C_DIS
   LIN {X 9.467, Y 4.636, Z 39.950} C_DIS
   LIN {X 9.407, Y 0.499, Z 39.950} C_DIS
   LIN {X 9.410, Y -3.593, Z 39.950} C_DIS
   LIN {X 9.110, Y -7.828, Z 39.950} C_DIS
   LIN {X 9.020, Y -9.189, Z 39.950} C_DIS
   LIN {X 8.919, Y -10.097, Z 39.950} C_DIS
   LIN {X 8.478, Y -13.836, Z 39.950} C_DIS
   LIN {X 7.893, Y -17.586, Z 39.950} C_DIS
   LIN {X 7.875, Y -17.689, Z 39.950} C_DIS
   LIN {X 7.339, Y -20.544, Z 39.950} C_DIS
   LIN {X 6.920, Y -22.504, Z 39.950} C_DIS
   LIN {X 6.649, Y -23.734, Z 39.950} C_DIS
   LIN {X 5.935, Y -25.437, Z 39.950} C_DIS
   LIN {X 5.504, Y -26.479, Z 39.950} C_DIS
   LIN {X 5.032, Y -27.011, Z 39.950} C_DIS
   LIN {X 3.105, Y -29.032, Z 39.950} C_DIS
   LIN {X 0.434, Y -30.273, Z 39.950} C_DIS
   LIN {X -0.214, Y -30.534, Z 39.950} C_DIS
   LIN {X -0.792, Y -30.550, Z 39.950} C_DIS
   LIN {X -3.284, Y -30.688, Z 39.950} C_DIS
   LIN {X -5.623, Y -29.906, Z 39.950} C_DIS
   LIN {X -6.701, Y -29.543, Z 39.950} C_DIS
   LIN {X -7.682, Y -28.733, Z 39.950} C_DIS
   LIN {X -8.992, Y -27.641, Z 39.950} C_DIS
   LIN {X -9.969, Y -25.857, Z 39.950} C_DIS
   LIN {X -10.783, Y -24.347, Z 39.950} C_DIS
   LIN {X -10.881, Y -23.024, Z 39.950} C_DIS
   LIN {X -11.075, Y -20.648, Z 39.950} C_DIS
   LIN {X -10.173, Y -17.782, Z 39.950} C_DIS
   LIN {X -10.124, Y -17.624, Z 39.950} C_DIS
   LIN {X -10.002, Y -17.369, Z 39.950} C_DIS
   LIN {X -8.527, Y -14.356, Z 39.950} C_DIS
   LIN {X -7.199, Y -11.257, Z 39.950} C_DIS
   LIN {X -6.978, Y -10.727, Z 39.950} C_DIS
   LIN {X -6.587, Y -9.618, Z 39.950} C_DIS
   LIN {X -5.412, Y -6.343, Z 39.950} C_DIS
   LIN {X -4.992, Y -4.966, Z 39.950} C_DIS
   LIN {X -4.177, Y -2.077, Z 39.950} C_DIS
   LIN {X -2.937, Y 3.795, Z 39.950} C_DIS
   LIN {X -2.841, Y 4.282, Z 39.950} C_DIS
   LIN {X -2.823, Y 4.501, Z 39.950} C_DIS
   LIN {X -1.964, Y 12.614, Z 39.950} C_DIS
   LIN {X -2.114, Y 16.272, Z 39.950} C_DIS
   LIN {X -2.142, Y 21.760, Z 39.950}
   LaserEnd_Ext()
   LIN {X -9.280, Y -25.028, Z 39.950}
   LaserStart_Ext()
   LIN {X -9.280, Y -18.275, Z 39.950}
   LaserEnd_Ext()
   LIN {X -8.280, Y -16.126, Z 39.950}
   LaserStart_Ext()
   LIN {X -8.280, Y -26.859, Z 39.950}
   LaserEnd_Ext()
   LIN {X -7.280, Y -27.767, Z 39.950}
   LaserStart_Ext()
   LIN {X -7.280, Y -24.663, Z 39.950}
   LaserEnd_Ext()
   LIN {X -7.280, Y -18.855, Z 39.950}
   LaserStart_Ext()
   LIN {X -7.280, Y -13.985, Z 39.950}
   LaserEnd_Ext()
   LIN {X -6.280, Y -11.650, Z 39.950}
   LaserStart_Ext()
   LIN {X -6.280, Y -17.574, Z 39.950}
   LaserEnd_Ext()
   LIN {X -6.280, Y -26.079, Z 39.950}
   LaserStart_Ext()
   LIN {X -6.280, Y -28.594, Z 39.950}
   LaserEnd_Ext()
   LIN {X -5.280, Y -28.966, Z 39.950}
   LaserStart_Ext()
   LIN {X -5.280, Y -26.755, Z 39.950}
   LaserEnd_Ext()
   LIN {X -5.280, Y -16.649, Z 39.950}
   LaserStart_Ext()
   LIN {X -5.280, Y -8.935, Z 39.950}
   LaserEnd_Ext()
   LIN {X -4.280, Y 41.181, Z 39.950}
   LaserStart_Ext()
   LIN {X -4.280, Y 38.116, Z 39.950}
   LaserEnd_Ext()
   LIN {X -4.280, Y -6.058, Z 39.950}
   LaserStart_Ext()
   LIN {X -4.280, Y -16.290, Z 39.950}
   LaserEnd_Ext()
   LIN {X -4.280, Y -27.359, Z 39.950}
   LaserStart_Ext()
   LIN {X -4.280, Y -29.301, Z 39.950}
   LaserEnd_Ext()
   LIN {X -3.280, Y -29.635, Z 39.950}
   LaserStart_Ext()
   LIN {X -3.280, Y -27.537, Z 39.950}
   LaserEnd_Ext()
   LIN {X -3.280, Y -15.989, Z 39.950}
   LaserStart_Ext()
   LIN {X -3.280, Y -2.581, Z 39.950}
   LaserEnd_Ext()
   LIN {X -3.280, Y 34.596, Z 39.950}
   LaserStart_Ext()
   LIN {X -3.280, Y 42.178, Z 39.950}
   LaserEnd_Ext()
   LIN {X -2.280, Y 42.580, Z 39.950}
   LaserStart_Ext()
   LIN {X -2.280, Y 30.172, Z 39.950}
   LaserEnd_Ext()
   LIN {X -2.280, Y 2.065, Z 39.950}
   LaserStart_Ext()
   LIN {X -2.280, Y -15.748, Z 39.950}
   LaserEnd_Ext()
   LIN {X -2.280, Y -27.712, Z 39.950}
   LaserStart_Ext()
   LIN {X -2.280, Y -29.631, Z 39.950}
   LaserEnd_Ext()
   LIN {X -1.280, Y -29.575, Z 39.950}
   LaserStart_Ext()
   LIN {X -1.280, Y -27.589, Z 39.950}
   LaserEnd_Ext()
   LIN {X -1.280, Y -15.906, Z 39.950}
   LaserStart_Ext()
   LIN {X -1.280, Y 9.578, Z 39.950}
   LaserEnd_Ext()
   LIN {X -1.280, Y 22.898, Z 39.950}
   LaserStart_Ext()
   LIN {X -1.280, Y 42.695, Z 39.950}
   LaserEnd_Ext()
   LIN {X -0.280, Y 42.365, Z 39.950}
   LaserStart_Ext()
   LIN {X -0.280, Y -16.072, Z 39.950}
   LaserEnd_Ext()
   LIN {X -0.280, Y -27.334, Z 39.950}
   LaserStart_Ext()
   LIN {X -0.280, Y -29.482, Z 39.950}
   LaserEnd_Ext()
   LIN {X 0.720, Y -29.038, Z 39.950}
   LaserStart_Ext()
   LIN {X 0.720, Y -26.995, Z 39.950}
   LaserEnd_Ext()
   LIN {X 0.720, Y -16.544, Z 39.950}
   LaserStart_Ext()
   LIN {X 0.720, Y 41.466, Z 39.950}
   LaserEnd_Ext()
   LIN {X 1.720, Y 39.231, Z 39.950}
   LaserStart_Ext()
   LIN {X 1.720, Y -17.224, Z 39.950}
   LaserEnd_Ext()
   LIN {X 1.720, Y -26.192, Z 39.950}
   LaserStart_Ext()
   LIN {X 1.720, Y -28.573, Z 39.950}
   LaserEnd_Ext()
   LIN {X 2.720, Y -27.987, Z 39.950}
   LaserStart_Ext()
   LIN {X 2.720, Y -25.137, Z 39.950}
   LaserEnd_Ext()
   LIN {X 2.720, Y -18.421, Z 39.950}
   LaserStart_Ext()
   LIN {X 2.720, Y 36.396, Z 39.950}
   LaserEnd_Ext()
   LIN {X 3.720, Y 33.274, Z 39.950}
   LaserStart_Ext()
   LIN {X 3.720, Y -20.398, Z 39.950}
   LaserEnd_Ext()
   LIN {X 3.720, Y -23.013, Z 39.950}
   LaserStart_Ext()
   LIN {X 3.720, Y -26.938, Z 39.950}
   LaserEnd_Ext()
   LIN {X 4.720, Y -25.759, Z 39.950}
   LaserStart_Ext()
   LIN {X 4.720, Y 29.763, Z 39.950}
   LaserEnd_Ext()
   LIN {X 5.720, Y 25.646, Z 39.950}
   LaserStart_Ext()
   LIN {X 5.720, Y -23.301, Z 39.950}
   LaserEnd_Ext()
   LIN {X 6.720, Y -18.421, Z 39.950}
   LaserStart_Ext()
   LIN {X 6.720, Y 20.480, Z 39.950}
   LaserEnd_Ext()
   LIN {X 7.720, Y 13.435, Z 39.950}
   LaserStart_Ext()
   LIN {X 7.720, Y -11.725, Z 39.950}
   LaserEnd_Ext()
   LIN {X 2.196, Y -19.364, Z 40.800}
   LaserStart_Ext()
   LIN {X 2.801, Y -20.458, Z 40.800} C_DIS
   LIN {X 2.826, Y -21.415, Z 40.800} C_DIS
   LIN {X 2.852, Y -22.634, Z 40.800} C_DIS
   LIN {X 2.456, Y -23.464, Z 40.800} C_DIS
   LIN {X 1.835, Y -24.810, Z 40.800} C_DIS
   LIN {X 0.409, Y -25.979, Z 40.800} C_DIS
   LIN {X 0.198, Y -26.149, Z 40.800} C_DIS
   LIN {X -0.258, Y -26.265, Z 40.800} C_DIS
   LIN {X -1.926, Y -26.694, Z 40.800} C_DIS
   LIN {X -2.951, Y -26.519, Z 40.800} C_DIS
   LIN {X -3.943, Y -26.347, Z 40.800} C_DIS
   LIN {X -5.040, Y -25.608, Z 40.800} C_DIS
   LIN {X -5.657, Y -25.195, Z 40.800} C_DIS
   LIN {X -6.000, Y -24.654, Z 40.800} C_DIS
   LIN {X -6.768, Y -23.433, Z 40.800} C_DIS
   LIN {X -6.955, Y -22.051, Z 40.800} C_DIS
   LIN {X -7.050, Y -21.365, Z 40.800} C_DIS
   LIN {X -6.781, Y -20.631, Z 40.800} C_DIS
   LIN {X -6.126, Y -18.806, Z 40.800} C_DIS
   LIN {X -4.853, Y -17.623, Z 40.800} C_DIS
   LIN {X -4.595, Y -17.396, Z 40.800} C_DIS
   LIN {X -4.162, Y -17.272, Z 40.800} C_DIS
   LIN {X -2.263, Y -16.697, Z 40.800} C_DIS
   LIN {X -1.062, Y -16.896, Z 40.800} C_DIS
   LIN {X -0.184, Y -17.038, Z 40.800} C_DIS
   LIN {X 0.687, Y -17.626, Z 40.800} C_DIS
   LIN {X 1.575, Y -18.230, Z 40.800} C_DIS
   LIN {X 2.196, Y -19.364, Z 40.800}
   LaserEnd_Ext()
   LIN {X 8.214, Y -15.831, Z 40.800}
   LaserStart_Ext()
   LIN {X 7.952, Y -17.562, Z 40.800} C_DIS
   LIN {X 7.735, Y -18.754, Z 40.800} C_DIS
   LIN {X 7.413, Y -20.473, Z 40.800} C_DIS
   LIN {X 6.741, Y -23.616, Z 40.800} C_DIS
   LIN {X 6.702, Y -23.730, Z 40.800} C_DIS
   LIN {X 5.596, Y -26.406, Z 40.800} C_DIS
   LIN {X 4.381, Y -27.773, Z 40.800} C_DIS
   LIN {X 3.328, Y -28.878, Z 40.800} C_DIS
   LIN {X 0.988, Y -29.965, Z 40.800} C_DIS
   LIN {X 0.023, Y -30.447, Z 40.800} C_DIS
   LIN {X -0.770, Y -30.514, Z 40.800} C_DIS
   LIN {X -3.152, Y -30.646, Z 40.800} C_DIS
   LIN {X -6.656, Y -29.474, Z 40.800} C_DIS
   LIN {X -8.902, Y -27.608, Z 40.800} C_DIS
   LIN {X -10.570, Y -24.560, Z 40.800} C_DIS
   LIN {X -10.701, Y -24.319, Z 40.800} C_DIS
   LIN {X -10.716, Y -24.107, Z 40.800} C_DIS
   LIN {X -11.001, Y -20.620, Z 40.800} C_DIS
   LIN {X -10.398, Y -18.703, Z 40.800} C_DIS
   LIN {X -10.057, Y -17.593, Z 40.800} C_DIS
   LIN {X -9.202, Y -15.816, Z 40.800} C_DIS
   LIN {X -8.426, Y -14.233, Z 40.800} C_DIS
   LIN {X -7.729, Y -12.604, Z 40.800} C_DIS
   LIN {X -6.916, Y -10.661, Z 40.800} C_DIS
   LIN {X -5.484, Y -6.593, Z 40.800} C_DIS
   LIN {X -5.283, Y -6.034, Z 40.800} C_DIS
   LIN {X -5.212, Y -5.799, Z 40.800} C_DIS
   LIN {X -4.126, Y -1.953, Z 40.800} C_DIS
   LIN {X -3.159, Y 2.626, Z 40.800} C_DIS
   LIN {X -2.830, Y 4.297, Z 40.800} C_DIS
   LIN {X -2.771, Y 5.046, Z 40.800} C_DIS
   LIN {X -1.969, Y 12.617, Z 40.800} C_DIS
   LIN {X -2.163, Y 17.365, Z 40.800} C_DIS
   LIN {X -2.187, Y 22.023, Z 40.800} C_DIS
   LIN {X -2.651, Y 25.641, Z 40.800} C_DIS
   LIN {X -2.865, Y 27.650, Z 40.800} C_DIS
   LIN {X -2.966, Y 28.185, Z 40.800} C_DIS
   LIN {X -3.452, Y 30.805, Z 40.800} C_DIS
   LIN {X -3.778, Y 32.234, Z 40.800} C_DIS
   LIN {X -4.100, Y 33.628, Z 40.800} C_DIS
   LIN {X -4.494, Y 35.093, Z 40.800} C_DIS
   LIN {X -4.714, Y 35.918, Z 40.800} C_DIS
   LIN {X -4.829, Y 36.307, Z 40.800} C_DIS
   LIN {X -5.170, Y 37.452, Z 40.800} C_DIS
   LIN {X -5.475, Y 38.428, Z 40.800} C_DIS
   LIN {X -5.544, Y 38.646, Z 40.800} C_DIS
   LIN {X -5.599, Y 39.056, Z 40.800} C_DIS
   LIN {X -5.744, Y 40.100, Z 40.800} C_DIS
   LIN {X -5.573, Y 40.881, Z 40.800} C_DIS
   LIN {X -5.425, Y 41.471, Z 40.800} C_DIS
   LIN {X -4.797, Y 42.321, Z 40.800} C_DIS
   LIN {X -4.381, Y 42.900, Z 40.800} C_DIS
   LIN {X -2.603, Y 43.608, Z 40.800} C_DIS
   LIN {X -1.959, Y 43.867, Z 40.800} C_DIS
   LIN {X -0.892, Y 43.677, Z 40.800} C_DIS
   LIN {X -0.239, Y 43.561, Z 40.800} C_DIS
   LIN {X 0.096, Y 43.325, Z 40.800} C_DIS
   LIN {X 1.184, Y 42.557, Z 40.800} C_DIS
   LIN {X 1.871, Y 41.447, Z 40.800} C_DIS
   LIN {X 1.959, Y 41.305, Z 40.800} C_DIS
   LIN {X 2.035, Y 41.104, Z 40.800} C_DIS
   LIN {X 2.506, Y 39.873, Z 40.800} C_DIS
   LIN {X 2.960, Y 38.625, Z 40.800} C_DIS
   LIN {X 3.265, Y 37.780, Z 40.800} C_DIS
   LIN {X 3.374, Y 37.462, Z 40.800} C_DIS
   LIN {X 4.162, Y 35.106, Z 40.800} C_DIS
   LIN {X 4.697, Y 33.411, Z 40.800} C_DIS
   LIN {X 5.157, Y 31.846, Z 40.800} C_DIS
   LIN {X 5.963, Y 28.943, Z 40.800} C_DIS
   LIN {X 6.723, Y 25.698, Z 40.800} C_DIS
   LIN {X 7.407, Y 22.657, Z 40.800} C_DIS
   LIN {X 8.018, Y 18.260, Z 40.800} C_DIS
   LIN {X 8.927, Y 12.238, Z 40.800} C_DIS
   LIN {X 9.313, Y 7.712, Z 40.800} C_DIS
   LIN {X 9.481, Y 4.721, Z 40.800} C_DIS
   LIN {X 9.440, Y 1.889, Z 40.800} C_DIS
   LIN {X 9.445, Y -3.505, Z 40.800} C_DIS
   LIN {X 9.334, Y -5.070, Z 40.800} C_DIS
   LIN {X 9.068, Y -9.102, Z 40.800} C_DIS
   LIN {X 8.768, Y -11.791, Z 40.800} C_DIS
   LIN {X 8.534, Y -13.780, Z 40.800} C_DIS
   LIN {X 8.214, Y -15.831, Z 40.800}
   LaserEnd_Ext()
   LIN {X -3.844, Y -29.360, Z 40.800}
   LaserStart_Ext()
   LIN {X -0.039, Y -29.360, Z 40.800}
   LaserEnd_Ext()
   LIN {X 2.069, Y -28.360, Z 40.800}
   LaserStart_Ext()
   LIN {X -6.438, Y -28.360, Z 40.800}
   LaserEnd_Ext()
   LIN {X -7.638, Y -27.360, Z 40.800}
   LaserStart_Ext()
   LIN {X -3.952, Y -27.360, Z 40.800}
   LaserEnd_Ext()
   LIN {X -0.502, Y -27.360, Z 40.800}
   LaserStart_Ext()
   LIN {X 3.393, Y -27.360, Z 40.800}
   LaserEnd_Ext()
   LIN {X 4.299, Y -26.360, Z 40.800}
   LaserStart_Ext()
   LIN {X 1.521, Y -26.360, Z 40.800}
   LaserEnd_Ext()
   LIN {X -5.714, Y -26.360, Z 40.800}
   LaserStart_Ext()
   LIN {X -8.445, Y -26.360, Z 40.800}
   LaserEnd_Ext()
   LIN {X -8.993, Y -25.360, Z 40.800}
   LaserStart_Ext()
   LIN {X -6.737, Y -25.360, Z 40.800}
   LaserEnd_Ext()
   LIN {X 2.669, Y -25.360, Z 40.800}
   LaserStart_Ext()
   LIN {X 4.946, Y -25.360, Z 40.800}
   LaserEnd_Ext()
   LIN {X 5.360, Y -24.360, Z 40.800}
   LaserStart_Ext()
   LIN {X 3.144, Y -24.360, Z 40.800}
   LaserEnd_Ext()
   LIN {X -7.366, Y -24.360, Z 40.800}
   LaserStart_Ext()
   LIN {X -9.540, Y -24.360, Z 40.800}
   LaserEnd_Ext()
   LIN {X -9.774, Y -23.360, Z 40.800}
   LaserStart_Ext()
   LIN {X -7.787, Y -23.360, Z 40.800}
   LaserEnd_Ext()
   LIN {X 3.613, Y -23.360, Z 40.800}
   LaserStart_Ext()
   LIN {X 5.773, Y -23.360, Z 40.800}
   LaserEnd_Ext()
   LIN {X 5.987, Y -22.360, Z 40.800}
   LaserStart_Ext()
   LIN {X 3.846, Y -22.360, Z 40.800}
   LaserEnd_Ext()
   LIN {X -7.922, Y -22.360, Z 40.800}
   LaserStart_Ext()
   LIN {X -9.856, Y -22.360, Z 40.800}
   LaserEnd_Ext()
   LIN {X -9.938, Y -21.360, Z 40.800}
   LaserStart_Ext()
   LIN {X -8.049, Y -21.360, Z 40.800}
   LaserEnd_Ext()
   LIN {X 3.825, Y -21.360, Z 40.800}
   LaserStart_Ext()
   LIN {X 6.200, Y -21.360, Z 40.800}
   LaserEnd_Ext()
   LIN {X 6.414, Y -20.360, Z 40.800}
   LaserStart_Ext()
   LIN {X 3.796, Y -20.360, Z 40.800}
   LaserEnd_Ext()
   LIN {X -7.747, Y -20.360, Z 40.800}
   LaserStart_Ext()
   LIN {X -9.871, Y -20.360, Z 40.800}
   LaserEnd_Ext()
   LIN {X -9.556, Y -19.360, Z 40.800}
   LaserStart_Ext()
   LIN {X -7.388, Y -19.360, Z 40.800}
   LaserEnd_Ext()
   LIN {X 3.337, Y -19.360, Z 40.800}
   LaserStart_Ext()
   LIN {X 6.604, Y -19.360, Z 40.800}
   LaserEnd_Ext()
   LIN {X 6.791, Y -18.360, Z 40.800}
   LaserStart_Ext()
   LIN {X 2.787, Y -18.360, Z 40.800}
   LaserEnd_Ext()
   LIN {X -7.020, Y -18.360, Z 40.800}
   LaserStart_Ext()
   LIN {X -9.247, Y -18.360, Z 40.800}
   LaserEnd_Ext()
   LIN {X -8.835, Y -17.360, Z 40.800}
   LaserStart_Ext()
   LIN {X -6.039, Y -17.360, Z 40.800}
   LaserEnd_Ext()
   LIN {X 2.074, Y -17.360, Z 40.800}
   LaserStart_Ext()
   LIN {X 6.972, Y -17.360, Z 40.800}
   LaserEnd_Ext()
   LIN {X 7.123, Y -16.360, Z 40.800}
   LaserStart_Ext()
   LIN {X 0.599, Y -16.360, Z 40.800}
   LaserEnd_Ext()
   LIN {X -4.609, Y -16.360, Z 40.800}
   LaserStart_Ext()
   LIN {X -8.354, Y -16.360, Z 40.800}
   LaserEnd_Ext()
   LIN {X -7.865, Y -15.360, Z 40.800}
   LaserStart_Ext()
   LIN {X 7.275, Y -15.360, Z 40.800}
   LaserEnd_Ext()
   LIN {X 7.431, Y -14.360, Z 40.800}
   LaserStart_Ext()
   LIN {X -7.393, Y -14.360, Z 40.800}
   LaserEnd_Ext()
   LIN {X -6.965, Y -13.360, Z 40.800}
   LaserStart_Ext()
   LIN {X 7.576, Y -13.360, Z 40.800}
   LaserEnd_Ext()
   LIN {X 7.694, Y -12.360, Z 40.800}
   LaserStart_Ext()
   LIN {X -6.543, Y -12.360, Z 40.800}
   LaserEnd_Ext()
   LIN {X -6.125, Y -11.360, Z 40.800}
   LaserStart_Ext()
   LIN {X 7.810, Y -11.360, Z 40.800}
   LaserEnd_Ext()
   LIN {X 7.922, Y -10.360, Z 40.800}
   LaserStart_Ext()
   LIN {X -5.750, Y -10.360, Z 40.800}
   LaserEnd_Ext()
   LIN {X -5.398, Y -9.360, Z 40.800}
   LaserStart_Ext()
   LIN {X 8.033, Y -9.360, Z 40.800}
   LaserEnd_Ext()
   LIN {X 8.115, Y -8.360, Z 40.800}
   LaserStart_Ext()
   LIN {X -5.046, Y -8.360, Z 40.800}
   LaserEnd_Ext()
   LIN {X -4.694, Y -7.360, Z 40.800}
   LaserStart_Ext()
   LIN {X 8.181, Y -7.360, Z 40.800}
   LaserEnd_Ext()
   LIN {X 8.247, Y -6.360, Z 40.800}
   LaserStart_Ext()
   LIN {X -4.338, Y -6.360, Z 40.800}
   LaserEnd_Ext()
   LIN {X -4.049, Y -5.360, Z 40.800}
   LaserStart_Ext()
   LIN {X 8.313, Y -5.360, Z 40.800}
   LaserEnd_Ext()
   LIN {X 8.382, Y -4.360, Z 40.800}
   LaserStart_Ext()
   LIN {X -3.766, Y -4.360, Z 40.800}
   LaserEnd_Ext()
   LIN {X -3.484, Y -3.360, Z 40.800}
   LaserStart_Ext()
   LIN {X 8.445, Y -3.360, Z 40.800}
   LaserEnd_Ext()
   LIN {X 8.444, Y -2.360, Z 40.800}
   LaserStart_Ext()
   LIN {X -3.202, Y -2.360, Z 40.800}
   LaserEnd_Ext()
   LIN {X -2.979, Y -1.360, Z 40.800}
   LaserStart_Ext()
   LIN {X 8.443, Y -1.360, Z 40.800}
   LaserEnd_Ext()
   LIN {X 8.442, Y -0.360, Z 40.800}
   LaserStart_Ext()
   LIN {X -2.768, Y -0.360, Z 40.800}
   LaserEnd_Ext()
   LIN {X -2.557, Y 0.640, Z 40.800}
   LaserStart_Ext()
   LIN {X 8.441, Y 0.640, Z 40.800}
   LaserEnd_Ext()
   LIN {X 8.440, Y 1.640, Z 40.800}
   LaserStart_Ext()
   LIN {X -2.345, Y 1.640, Z 40.800}
   LaserEnd_Ext()
   LIN {X -2.137, Y 2.640, Z 40.800}
   LaserStart_Ext()
   LIN {X 8.451, Y 2.640, Z 40.800}
   LaserEnd_Ext()
   LIN {X 8.465, Y 3.640, Z 40.800}
   LaserStart_Ext()
   LIN {X -1.940, Y 3.640, Z 40.800}
   LaserEnd_Ext()
   LIN {X -1.800, Y 4.640, Z 40.800}
   LaserStart_Ext()
   LIN {X 8.480, Y 4.640, Z 40.800}
   LaserEnd_Ext()
   LIN {X 8.428, Y 5.640, Z 40.800}
   LaserStart_Ext()
   LIN {X -1.702, Y 5.640, Z 40.800}
   LaserEnd_Ext()
   LIN {X -1.596, Y 6.640, Z 40.800}
   LaserStart_Ext()
   LIN {X 8.372, Y 6.640, Z 40.800}
   LaserEnd_Ext()
   LIN {X 8.315, Y 7.640, Z 40.800}
   LaserStart_Ext()
   LIN {X -1.490, Y 7.640, Z 40.800}
   LaserEnd_Ext()
   LIN {X -1.384, Y 8.640, Z 40.800}
   LaserStart_Ext()
   LIN {X 8.230, Y 8.640, Z 40.800}
   LaserEnd_Ext()
   LIN {X 8.145, Y 9.640, Z 40.800}
   LaserStart_Ext()
   LIN {X -1.278, Y 9.640, Z 40.800}
   LaserEnd_Ext()
   LIN {X -1.172, Y 10.640, Z 40.800}
   LaserStart_Ext()
   LIN {X 8.060, Y 10.640, Z 40.800}
   LaserEnd_Ext()
   LIN {X 7.975, Y 11.640, Z 40.800}
   LaserStart_Ext()
   LIN {X -1.067, Y 11.640, Z 40.800}
   LaserEnd_Ext()
   LIN {X -0.970, Y 12.640, Z 40.800}
   LaserStart_Ext()
   LIN {X 7.855, Y 12.640, Z 40.800}
   LaserEnd_Ext()
   LIN {X 7.704, Y 13.640, Z 40.800}
   LaserStart_Ext()
   LIN {X -1.010, Y 13.640, Z 40.800}
   LaserEnd_Ext()
   LIN {X -1.051, Y 14.640, Z 40.800}
   LaserStart_Ext()
   LIN {X 7.553, Y 14.640, Z 40.800}
   LaserEnd_Ext()
   LIN {X 7.402, Y 15.640, Z 40.800}
   LaserStart_Ext()
   LIN {X -1.092, Y 15.640, Z 40.800}
   LaserEnd_Ext()
   LIN {X -1.133, Y 16.640, Z 40.800}
   LaserStart_Ext()
   LIN {X 7.252, Y 16.640, Z 40.800}
   LaserEnd_Ext()
   LIN {X 7.101, Y 17.640, Z 40.800}
   LaserStart_Ext()
   LIN {X -1.165, Y 17.640, Z 40.800}
   LaserEnd_Ext()
   LIN {X -1.170, Y 18.640, Z 40.800}
   LaserStart_Ext()
   LIN {X 6.956, Y 18.640, Z 40.800}
   LaserEnd_Ext()
   LIN {X 6.817, Y 19.640, Z 40.800}
   LaserStart_Ext()
   LIN {X -1.175, Y 19.640, Z 40.800}
   LaserEnd_Ext()
   LIN {X -1.180, Y 20.640, Z 40.800}
   LaserStart_Ext()
   LIN {X 6.678, Y 20.640, Z 40.800}
   LaserEnd_Ext()
   LIN {X 6.539, Y 21.640, Z 40.800}
   LaserStart_Ext()
   LIN {X -1.185, Y 21.640, Z 40.800}
   LaserEnd_Ext()
   LIN {X -1.258, Y 22.640, Z 40.800}
   LaserStart_Ext()
   LIN {X 6.386, Y 22.640, Z 40.800}
   LaserEnd_Ext()
   LIN {X 6.161, Y 23.640, Z 40.800}
   LaserStart_Ext()
   LIN {X -1.386, Y 23.640, Z 40.800}
   LaserEnd_Ext()
   LIN {X -1.514, Y 24.640, Z 40.800}
   LaserStart_Ext()
   LIN {X 5.936, Y 24.640, Z 40.800}
   LaserEnd_Ext()
   LIN {X 5.710, Y 25.640, Z 40.800}
   LaserStart_Ext()
   LIN {X -1.642, Y 25.640, Z 40.800}
   LaserEnd_Ext()
   LIN {X -1.752, Y 26.640, Z 40.800}
   LaserStart_Ext()
   LIN {X 5.475, Y 26.640, Z 40.800}
   LaserEnd_Ext()
   LIN {X 5.241, Y 27.640, Z 40.800}
   LaserStart_Ext()
   LIN {X -1.859, Y 27.640, Z 40.800}
   LaserEnd_Ext()
   LIN {X -2.033, Y 28.640, Z 40.800}
   LaserStart_Ext()
   LIN {X 5.007, Y 28.640, Z 40.800}
   LaserEnd_Ext()
   LIN {X 4.731, Y 29.640, Z 40.800}
   LaserStart_Ext()
   LIN {X -2.219, Y 29.640, Z 40.800}
   LaserEnd_Ext()
   LIN {X -2.405, Y 30.640, Z 40.800}
   LaserStart_Ext()
   LIN {X 4.454, Y 30.640, Z 40.800}
   LaserEnd_Ext()
   LIN {X 4.175, Y 31.640, Z 40.800}
   LaserStart_Ext()
   LIN {X -2.617, Y 31.640, Z 40.800}
   LaserEnd_Ext()
   LIN {X -2.846, Y 32.640, Z 40.800}
   LaserStart_Ext()
   LIN {X 3.881, Y 32.640, Z 40.800}
   LaserEnd_Ext()
   LIN {X 3.576, Y 33.640, Z 40.800}
   LaserStart_Ext()
   LIN {X -3.077, Y 33.640, Z 40.800}
   LaserEnd_Ext()
   LIN {X -3.337, Y 34.640, Z 40.800}
   LaserStart_Ext()
   LIN {X 3.260, Y 34.640, Z 40.800}
   LaserEnd_Ext()
   LIN {X 2.929, Y 35.640, Z 40.800}
   LaserStart_Ext()
   LIN {X -3.605, Y 35.640, Z 40.800}
   LaserEnd_Ext()
   LIN {X -3.884, Y 36.640, Z 40.800}
   LaserStart_Ext()
   LIN {X 2.594, Y 36.640, Z 40.800}
   LaserEnd_Ext()
   LIN {X 2.252, Y 37.640, Z 40.800}
   LaserStart_Ext()
   LIN {X -4.182, Y 37.640, Z 40.800}
   LaserEnd_Ext()
   LIN {X -4.494, Y 38.640, Z 40.800}
   LaserStart_Ext()
   LIN {X 1.890, Y 38.640, Z 40.800}
   LaserEnd_Ext()
   LIN {X 1.524, Y 39.640, Z 40.800}
   LaserStart_Ext()
   LIN {X -4.671, Y 39.640, Z 40.800}
   LaserEnd_Ext()
   LIN {X -4.602, Y 40.640, Z 40.800}
   LaserStart_Ext()
   LIN {X 1.142, Y 40.640, Z 40.800}
   LaserEnd_Ext()
   LIN {X 0.575, Y 41.640, Z 40.800}
   LaserStart_Ext()
   LIN {X -4.056, Y 41.640, Z 40.800}
   LaserEnd_Ext()
   LIN {X -2.331, Y 42.640, Z 40.800}
   LaserStart_Ext()
   LIN {X -0.773, Y 42.640, Z 40.800}
   LaserEnd_Ext()
   LIN {X -6.975, Y -21.328, Z 41.650}
   LaserStart_Ext()
   LIN {X -6.151, Y -19.080, Z 41.650} C_DIS
   LIN {X -6.021, Y -18.717, Z 41.650} C_DIS
   LIN {X -5.767, Y -18.481, Z 41.650} C_DIS
   LIN {X -4.394, Y -17.279, Z 41.650} C_DIS
   LIN {X -2.259, Y -16.665, Z 41.650} C_DIS
   LIN {X -2.116, Y -16.662, Z 41.650} C_DIS
   LIN {X -0.118, Y -16.985, Z 41.650} C_DIS
   LIN {X 1.314, Y -17.952, Z 41.650} C_DIS
   LIN {X 1.643, Y -18.173, Z 41.650} C_DIS
   LIN {X 1.894, Y -18.622, Z 41.650} C_DIS
   LIN {X 2.875, Y -20.397, Z 41.650} C_DIS
   LIN {X 2.925, Y -22.355, Z 41.650} C_DIS
   LIN {X 2.931, Y -22.573, Z 41.650} C_DIS
   LIN {X 2.661, Y -23.163, Z 41.650} C_DIS
   LIN {X 1.939, Y -24.727, Z 41.650} C_DIS
   LIN {X 1.443, Y -25.133, Z 41.650} C_DIS
   LIN {X 0.271, Y -26.101, Z 41.650} C_DIS
   LIN {X -1.837, Y -26.644, Z 41.650} C_DIS
   LIN {X -3.453, Y -26.370, Z 41.650} C_DIS
   LIN {X -3.855, Y -26.302, Z 41.650} C_DIS
   LIN {X -4.115, Y -26.130, Z 41.650} C_DIS
   LIN {X -5.573, Y -25.154, Z 41.650} C_DIS
   LIN {X -6.668, Y -23.426, Z 41.650} C_DIS
   LIN {X -6.975, Y -21.328, Z 41.650}
   LaserEnd_Ext()
   LIN {X -4.365, Y 34.461, Z 41.650}
   LaserStart_Ext()
   LIN {X -4.772, Y 35.961, Z 41.650} C_DIS
   LIN {X -5.170, Y 37.286, Z 41.650} C_DIS
   LIN {X -5.232, Y 37.493, Z 41.650} C_DIS
   LIN {X -5.609, Y 38.686, Z 41.650} C_DIS
   LIN {X -5.751, Y 39.743, Z 41.650} C_DIS
   LIN {X -5.811, Y 40.163, Z 41.650} C_DIS
   LIN {X -5.682, Y 40.655, Z 41.650} C_DIS
   LIN {X -5.430, Y 41.654, Z 41.650} C_DIS
   LIN {X -4.878, Y 42.400, Z 41.650} C_DIS
   LIN {X -4.438, Y 42.958, Z 41.650} C_DIS
   LIN {X -2.036, Y 43.916, Z 41.650} C_DIS
   LIN {X -1.320, Y 43.792, Z 41.650} C_DIS
   LIN {X -0.316, Y 43.614, Z 41.650} C_DIS
   LIN {X 0.980, Y 42.704, Z 41.650} C_DIS
   LIN {X 1.110, Y 42.614, Z 41.650} C_DIS
   LIN {X 1.888, Y 41.364, Z 41.650} C_DIS
   LIN {X 2.306, Y 40.278, Z 41.650} C_DIS
   LIN {X 2.424, Y 39.969, Z 41.650} C_DIS
   LIN {X 2.733, Y 39.120, Z 41.650} C_DIS
   LIN {X 3.237, Y 37.742, Z 41.650} C_DIS
   LIN {X 3.348, Y 37.424, Z 41.650} C_DIS
   LIN {X 3.870, Y 35.845, Z 41.650} C_DIS
   LIN {X 4.387, Y 34.300, Z 41.650} C_DIS
   LIN {X 4.537, Y 33.825, Z 41.650} C_DIS
   LIN {X 5.393, Y 30.912, Z 41.650} C_DIS
   LIN {X 5.911, Y 29.048, Z 41.650} C_DIS
   LIN {X 7.124, Y 23.871, Z 41.650} C_DIS
   LIN {X 7.372, Y 22.767, Z 41.650} C_DIS
   LIN {X 7.594, Y 21.169, Z 41.650} C_DIS
   LIN {X 8.865, Y 12.748, Z 41.650} C_DIS
   LIN {X 9.405, Y 6.417, Z 41.650} C_DIS
   LIN {X 9.496, Y 4.806, Z 41.650} C_DIS
   LIN {X 9.473, Y 3.279, Z 41.650} C_DIS
   LIN {X 9.477, Y -1.268, Z 41.650} C_DIS
   LIN {X 9.479, Y -3.420, Z 41.650} C_DIS
   LIN {X 9.427, Y -4.298, Z 41.650} C_DIS
   LIN {X 9.116, Y -9.015, Z 41.650} C_DIS
   LIN {X 8.617, Y -13.486, Z 41.650} C_DIS
   LIN {X 8.589, Y -13.725, Z 41.650} C_DIS
   LIN {X 8.551, Y -13.971, Z 41.650} C_DIS
   LIN {X 8.019, Y -17.489, Z 41.650} C_DIS
   LIN {X 7.578, Y -19.911, Z 41.650} C_DIS
   LIN {X 7.486, Y -20.402, Z 41.650} C_DIS
   LIN {X 7.286, Y -21.340, Z 41.650} C_DIS
   LIN {X 6.811, Y -23.594, Z 41.650} C_DIS
   LIN {X 6.363, Y -24.699, Z 41.650} C_DIS
   LIN {X 5.687, Y -26.333, Z 41.650} C_DIS
   LIN {X 3.731, Y -28.534, Z 41.650} C_DIS
   LIN {X 3.551, Y -28.723, Z 41.650} C_DIS
   LIN {X 3.151, Y -28.909, Z 41.650} C_DIS
   LIN {X 0.259, Y -30.354, Z 41.650} C_DIS
   LIN {X -2.117, Y -30.554, Z 41.650} C_DIS
   LIN {X -3.019, Y -30.604, Z 41.650} C_DIS
   LIN {X -4.346, Y -30.160, Z 41.650} C_DIS
   LIN {X -6.574, Y -29.431, Z 41.650} C_DIS
   LIN {X -7.396, Y -28.756, Z 41.650} C_DIS
   LIN {X -8.811, Y -27.575, Z 41.650} C_DIS
   LIN {X -10.041, Y -25.330, Z 41.650} C_DIS
   LIN {X -10.618, Y -24.290, Z 41.650} C_DIS
   LIN {X -10.759, Y -22.656, Z 41.650} C_DIS
   LIN {X -10.928, Y -20.592, Z 41.650} C_DIS
   LIN {X -10.623, Y -19.623, Z 41.650} C_DIS
   LIN {X -9.990, Y -17.563, Z 41.650} C_DIS
   LIN {X -8.401, Y -14.263, Z 41.650} C_DIS
   LIN {X -8.326, Y -14.109, Z 41.650} C_DIS
   LIN {X -8.258, Y -13.950, Z 41.650} C_DIS
   LIN {X -6.855, Y -10.595, Z 41.650} C_DIS
   LIN {X -5.619, Y -7.085, Z 41.650} C_DIS
   LIN {X -5.242, Y -5.995, Z 41.650} C_DIS
   LIN {X -4.945, Y -4.909, Z 41.650} C_DIS
   LIN {X -4.076, Y -1.828, Z 41.650} C_DIS
   LIN {X -3.382, Y 1.458, Z 41.650} C_DIS
   LIN {X -2.819, Y 4.311, Z 41.650} C_DIS
   LIN {X -2.718, Y 5.591, Z 41.650} C_DIS
   LIN {X -1.973, Y 12.620, Z 41.650} C_DIS
   LIN {X -2.213, Y 18.459, Z 41.650} C_DIS
   LIN {X -2.233, Y 22.287, Z 41.650} C_DIS
   LIN {X -2.799, Y 26.715, Z 41.650} C_DIS
   LIN {X -2.904, Y 27.697, Z 41.650} C_DIS
   LIN {X -3.323, Y 29.928, Z 41.650} C_DIS
   LIN {X -3.499, Y 30.851, Z 41.650} C_DIS
   LIN {X -3.846, Y 32.344, Z 41.650} C_DIS
   LIN {X -4.153, Y 33.672, Z 41.650} C_DIS
   LIN {X -4.365, Y 34.461, Z 41.650}
   LaserEnd_Ext()
   LIN {X 7.602, Y -13.558, Z 41.650}
   LaserStart_Ext()
   LIN {X 7.602, Y 14.418, Z 41.650}
   LaserEnd_Ext()
   LIN {X 6.602, Y 21.046, Z 41.650}
   LaserStart_Ext()
   LIN {X 6.602, Y -19.692, Z 41.650}
   LaserEnd_Ext()
   LIN {X 5.602, Y -23.915, Z 41.650}
   LaserStart_Ext()
   LIN {X 5.602, Y 25.983, Z 41.650}
   LaserEnd_Ext()
   LIN {X 4.602, Y 30.024, Z 41.650}
   LaserStart_Ext()
   LIN {X 4.602, Y -26.049, Z 41.650}
   LaserEnd_Ext()
   LIN {X 3.602, Y -27.174, Z 41.650}
   LaserStart_Ext()
   LIN {X 3.602, Y -23.509, Z 41.650}
   LaserEnd_Ext()
   LIN {X 3.602, Y -19.645, Z 41.650}
   LaserStart_Ext()
   LIN {X 3.602, Y 33.460, Z 41.650}
   LaserEnd_Ext()
   LIN {X 2.602, Y 36.495, Z 41.650}
   LaserStart_Ext()
   LIN {X 2.602, Y -17.839, Z 41.650}
   LaserEnd_Ext()
   LIN {X 2.602, Y -25.474, Z 41.650}
   LaserStart_Ext()
   LIN {X 2.602, Y -28.065, Z 41.650}
   LaserEnd_Ext()
   LIN {X 1.602, Y -28.565, Z 41.650}
   LaserStart_Ext()
   LIN {X 1.602, Y -26.299, Z 41.650}
   LaserEnd_Ext()
   LIN {X 1.602, Y -16.940, Z 41.650}
   LaserStart_Ext()
   LIN {X 1.602, Y 39.304, Z 41.650}
   LaserEnd_Ext()
   LIN {X 0.602, Y 41.537, Z 41.650}
   LaserStart_Ext()
   LIN {X 0.602, Y -16.264, Z 41.650}
   LaserEnd_Ext()
   LIN {X 0.602, Y -27.044, Z 41.650}
   LaserStart_Ext()
   LIN {X 0.602, Y -29.065, Z 41.650}
   LaserEnd_Ext()
   LIN {X -0.398, Y -29.406, Z 41.650}
   LaserStart_Ext()
   LIN {X -0.398, Y -27.307, Z 41.650}
   LaserEnd_Ext()
   LIN {X -0.398, Y -15.927, Z 41.650}
   LaserStart_Ext()
   LIN {X -0.398, Y 42.450, Z 41.650}
   LaserEnd_Ext()
   LIN {X -1.398, Y 42.790, Z 41.650}
   LaserStart_Ext()
   LIN {X -1.398, Y 23.644, Z 41.650}
   LaserEnd_Ext()
   LIN {X -1.398, Y 8.558, Z 41.650}
   LaserStart_Ext()
   LIN {X -1.398, Y -15.765, Z 41.650}
   LaserEnd_Ext()
   LIN {X -1.398, Y -27.564, Z 41.650}
   LaserStart_Ext()
   LIN {X -1.398, Y -29.490, Z 41.650}
   LaserEnd_Ext()
   LIN {X -2.398, Y -29.568, Z 41.650}
   LaserStart_Ext()
   LIN {X -2.398, Y -27.563, Z 41.650}
   LaserEnd_Ext()
   LIN {X -2.398, Y -15.671, Z 41.650}
   LaserStart_Ext()
   LIN {X -2.398, Y 1.277, Z 41.650}
   LaserEnd_Ext()
   LIN {X -2.398, Y 30.417, Z 41.650}
   LaserStart_Ext()
   LIN {X -2.398, Y 42.695, Z 41.650}
   LaserEnd_Ext()
   LIN {X -3.398, Y 42.296, Z 41.650}
   LaserStart_Ext()
   LIN {X -3.398, Y 34.715, Z 41.650}
   LaserEnd_Ext()
   LIN {X -3.398, Y -3.109, Z 41.650}
   LaserStart_Ext()
   LIN {X -3.398, Y -15.952, Z 41.650}
   LaserEnd_Ext()
   LIN {X -3.398, Y -27.393, Z 41.650}
   LaserStart_Ext()
   LIN {X -3.398, Y -29.423, Z 41.650}
   LaserEnd_Ext()
   LIN {X -4.398, Y -29.091, Z 41.650}
   LaserStart_Ext()
   LIN {X -4.398, Y -27.141, Z 41.650}
   LaserEnd_Ext()
   LIN {X -4.398, Y -16.239, Z 41.650}
   LaserStart_Ext()
   LIN {X -4.398, Y -6.614, Z 41.650}
   LaserEnd_Ext()
   LIN {X -4.398, Y 38.175, Z 41.650}
   LaserStart_Ext()
   LIN {X -4.398, Y 41.368, Z 41.650}
   LaserEnd_Ext()
   LIN {X -5.398, Y -9.469, Z 41.650}
   LaserStart_Ext()
   LIN {X -5.398, Y -16.829, Z 41.650}
   LaserEnd_Ext()
   LIN {X -5.398, Y -26.474, Z 41.650}
   LaserStart_Ext()
   LIN {X -5.398, Y -28.764, Z 41.650}
   LaserEnd_Ext()
   LIN {X -6.398, Y -28.281, Z 41.650}
   LaserStart_Ext()
   LIN {X -6.398, Y -25.717, Z 41.650}
   LaserEnd_Ext()
   LIN {X -6.398, Y -17.704, Z 41.650}
   LaserStart_Ext()
   LIN {X -6.398, Y -12.095, Z 41.650}
   LaserEnd_Ext()
   LIN {X -7.398, Y -14.482, Z 41.650}
   LaserStart_Ext()
   LIN {X -7.398, Y -19.577, Z 41.650}
   LaserEnd_Ext()
   LIN {X -7.398, Y -24.141, Z 41.650}
   LaserStart_Ext()
   LIN {X -7.398, Y -27.452, Z 41.650}
   LaserEnd_Ext()
   LIN {X -8.398, Y -26.248, Z 41.650}
   LaserStart_Ext()
   LIN {X -8.398, Y -16.561, Z 41.650}
   LaserEnd_Ext()
   LIN {X -9.398, Y -19.041, Z 41.650}
   LaserStart_Ext()
   LIN {X -9.398, Y -24.427, Z 41.650}
   LaserEnd_Ext()
   LIN {X 3.010, Y -22.512, Z 42.500}
   LaserStart_Ext()
   LIN {X 2.301, Y -24.059, Z 42.500} C_DIS
   LIN {X 2.017, Y -24.677, Z 42.500} C_DIS
   LIN {X 1.351, Y -25.222, Z 42.500} C_DIS
   LIN {X 0.340, Y -26.056, Z 42.500} C_DIS
   LIN {X -1.749, Y -26.595, Z 42.500} C_DIS
   LIN {X -1.865, Y -26.576, Z 42.500} C_DIS
   LIN {X -3.768, Y -26.257, Z 42.500} C_DIS
   LIN {X -5.172, Y -25.325, Z 42.500} C_DIS
   LIN {X -5.488, Y -25.114, Z 42.500} C_DIS
   LIN {X -5.725, Y -24.740, Z 42.500} C_DIS
   LIN {X -6.607, Y -23.357, Z 42.500} C_DIS
   LIN {X -6.825, Y -21.824, Z 42.500} C_DIS
   LIN {X -6.899, Y -21.291, Z 42.500} C_DIS
   LIN {X -6.590, Y -20.447, Z 42.500} C_DIS
   LIN {X -5.915, Y -18.628, Z 42.500} C_DIS
   LIN {X -4.947, Y -17.821, Z 42.500} C_DIS
   LIN {X -4.194, Y -17.161, Z 42.500} C_DIS
   LIN {X -3.367, Y -16.923, Z 42.500} C_DIS
   LIN {X -2.129, Y -16.600, Z 42.500} C_DIS
   LIN {X -0.482, Y -16.862, Z 42.500} C_DIS
   LIN {X -0.053, Y -16.931, Z 42.500} C_DIS
   LIN {X 0.255, Y -17.139, Z 42.500} C_DIS
   LIN {X 1.712, Y -18.115, Z 42.500} C_DIS
   LIN {X 2.821, Y -20.106, Z 42.500} C_DIS
   LIN {X 2.949, Y -20.337, Z 42.500} C_DIS
   LIN {X 2.955, Y -20.592, Z 42.500} C_DIS
   LIN {X 3.010, Y -22.512, Z 42.500}
   LaserEnd_Ext()
   LIN {X -2.262, Y 19.552, Z 42.500}
   LaserStart_Ext()
   LIN {X -2.278, Y 22.550, Z 42.500} C_DIS
   LIN {X -2.936, Y 27.690, Z 42.500} C_DIS
   LIN {X -2.956, Y 27.805, Z 42.500} C_DIS
   LIN {X -2.980, Y 27.936, Z 42.500} C_DIS
   LIN {X -3.545, Y 30.896, Z 42.500} C_DIS
   LIN {X -3.882, Y 32.344, Z 42.500} C_DIS
   LIN {X -4.206, Y 33.715, Z 42.500} C_DIS
   LIN {X -4.646, Y 35.323, Z 42.500} C_DIS
   LIN {X -4.830, Y 36.003, Z 42.500} C_DIS
   LIN {X -4.938, Y 36.362, Z 42.500} C_DIS
   LIN {X -5.293, Y 37.535, Z 42.500} C_DIS
   LIN {X -5.621, Y 38.564, Z 42.500} C_DIS
   LIN {X -5.674, Y 38.727, Z 42.500} C_DIS
   LIN {X -5.707, Y 38.941, Z 42.500} C_DIS
   LIN {X -5.881, Y 40.151, Z 42.500} C_DIS
   LIN {X -5.523, Y 41.515, Z 42.500} C_DIS
   LIN {X -5.449, Y 41.808, Z 42.500} C_DIS
   LIN {X -5.199, Y 42.126, Z 42.500} C_DIS
   LIN {X -4.497, Y 43.014, Z 42.500} C_DIS
   LIN {X -2.113, Y 43.965, Z 42.500} C_DIS
   LIN {X -0.948, Y 43.762, Z 42.500} C_DIS
   LIN {X -0.392, Y 43.667, Z 42.500} C_DIS
   LIN {X -0.097, Y 43.462, Z 42.500} C_DIS
   LIN {X 1.036, Y 42.670, Z 42.500} C_DIS
   LIN {X 1.795, Y 41.457, Z 42.500} C_DIS
   LIN {X 2.353, Y 40.037, Z 42.500} C_DIS
   LIN {X 2.850, Y 38.690, Z 42.500} C_DIS
   LIN {X 3.168, Y 37.822, Z 42.500} C_DIS
   LIN {X 3.562, Y 36.689, Z 42.500} C_DIS
   LIN {X 4.198, Y 34.770, Z 42.500} C_DIS
   LIN {X 4.359, Y 34.276, Z 42.500} C_DIS
   LIN {X 4.398, Y 34.156, Z 42.500} C_DIS
   LIN {X 4.495, Y 33.861, Z 42.500} C_DIS
   LIN {X 5.060, Y 31.918, Z 42.500} C_DIS
   LIN {X 5.630, Y 29.977, Z 42.500} C_DIS
   LIN {X 5.859, Y 29.153, Z 42.500} C_DIS
   LIN {X 6.813, Y 25.082, Z 42.500} C_DIS
   LIN {X 7.307, Y 23.000, Z 42.500} C_DIS
   LIN {X 7.401, Y 22.552, Z 42.500} C_DIS
   LIN {X 8.804, Y 13.257, Z 42.500} C_DIS
   LIN {X 9.497, Y 5.123, Z 42.500} C_DIS
   LIN {X 9.510, Y 4.890, Z 42.500} C_DIS
   LIN {X 9.507, Y 4.670, Z 42.500} C_DIS
   LIN {X 9.507, Y 4.012, Z 42.500} C_DIS
   LIN {X 9.513, Y -3.340, Z 42.500} C_DIS
   LIN {X 9.335, Y -6.340, Z 42.500} C_DIS
   LIN {X 9.164, Y -8.929, Z 42.500} C_DIS
   LIN {X 8.857, Y -11.686, Z 42.500} C_DIS
   LIN {X 8.647, Y -13.653, Z 42.500} C_DIS
   LIN {X 8.489, Y -14.750, Z 42.500} C_DIS
   LIN {X 8.086, Y -17.417, Z 42.500} C_DIS
   LIN {X 7.674, Y -19.682, Z 42.500} C_DIS
   LIN {X 7.560, Y -20.330, Z 42.500} C_DIS
   LIN {X 7.415, Y -21.043, Z 42.500} C_DIS
   LIN {X 6.893, Y -23.524, Z 42.500} C_DIS
   LIN {X 5.977, Y -25.780, Z 42.500} C_DIS
   LIN {X 5.778, Y -26.260, Z 42.500} C_DIS
   LIN {X 5.054, Y -27.075, Z 42.500} C_DIS
   LIN {X 3.678, Y -28.636, Z 42.500} C_DIS
   LIN {X 2.677, Y -29.171, Z 42.500} C_DIS
   LIN {X 0.495, Y -30.261, Z 42.500} C_DIS
   LIN {X -2.179, Y -30.486, Z 42.500} C_DIS
   LIN {X -2.936, Y -30.555, Z 42.500} C_DIS
   LIN {X -3.486, Y -30.372, Z 42.500} C_DIS
   LIN {X -6.480, Y -29.393, Z 42.500} C_DIS
   LIN {X -8.118, Y -28.045, Z 42.500} C_DIS
   LIN {X -8.721, Y -27.542, Z 42.500} C_DIS
   LIN {X -9.245, Y -26.586, Z 42.500} C_DIS
   LIN {X -10.535, Y -24.261, Z 42.500} C_DIS
   LIN {X -10.850, Y -20.608, Z 42.500} C_DIS
   LIN {X -9.923, Y -17.533, Z 42.500} C_DIS
   LIN {X -8.772, Y -15.140, Z 42.500} C_DIS
   LIN {X -8.263, Y -14.065, Z 42.500} C_DIS
   LIN {X -7.687, Y -12.666, Z 42.500} C_DIS
   LIN {X -6.793, Y -10.529, Z 42.500} C_DIS
   LIN {X -6.074, Y -8.487, Z 42.500} C_DIS
   LIN {X -5.224, Y -6.024, Z 42.500} C_DIS
   LIN {X -4.552, Y -3.572, Z 42.500} C_DIS
   LIN {X -4.025, Y -1.704, Z 42.500} C_DIS
   LIN {X -3.604, Y 0.289, Z 42.500} C_DIS
   LIN {X -2.809, Y 4.325, Z 42.500} C_DIS
   LIN {X -2.665, Y 6.136, Z 42.500} C_DIS
   LIN {X -1.978, Y 12.624, Z 42.500} C_DIS
   LIN {X -2.262, Y 19.552, Z 42.500}
   LaserEnd_Ext()
   LIN {X -0.497, Y 42.522, Z 42.500}
   LaserStart_Ext()
   LIN {X -3.032, Y 42.522, Z 42.500}
   LaserEnd_Ext()
   LIN {X -4.401, Y 41.522, Z 42.500}
   LaserStart_Ext()
   LIN {X 0.575, Y 41.522, Z 42.500}
   LaserEnd_Ext()
   LIN {X 1.093, Y 40.522, Z 42.500}
   LaserStart_Ext()
   LIN {X -4.750, Y 40.522, Z 42.500}
   LaserEnd_Ext()
   LIN {X -4.780, Y 39.522, Z 42.500}
   LaserStart_Ext()
   LIN {X 1.478, Y 39.522, Z 42.500}
   LaserEnd_Ext()
   LIN {X 1.847, Y 38.522, Z 42.500}
   LaserStart_Ext()
   LIN {X -4.558, Y 38.522, Z 42.500}
   LaserEnd_Ext()
   LIN {X -4.245, Y 37.522, Z 42.500}
   LaserStart_Ext()
   LIN {X 2.213, Y 37.522, Z 42.500}
   LaserEnd_Ext()
   LIN {X 2.562, Y 36.522, Z 42.500}
   LaserStart_Ext()
   LIN {X -3.942, Y 36.522, Z 42.500}
   LaserEnd_Ext()
   LIN {X -3.663, Y 35.522, Z 42.500}
   LaserStart_Ext()
   LIN {X 2.895, Y 35.522, Z 42.500}
   LaserEnd_Ext()
   LIN {X 3.227, Y 34.522, Z 42.500}
   LaserStart_Ext()
   LIN {X -3.390, Y 34.522, Z 42.500}
   LaserEnd_Ext()
   LIN {X -3.133, Y 33.522, Z 42.500}
   LaserStart_Ext()
   LIN {X 3.552, Y 33.522, Z 42.500}
   LaserEnd_Ext()
   LIN {X 3.843, Y 32.522, Z 42.500}
   LaserStart_Ext()
   LIN {X -2.897, Y 32.522, Z 42.500}
   LaserEnd_Ext()
   LIN {X -2.664, Y 31.522, Z 42.500}
   LaserStart_Ext()
   LIN {X 4.134, Y 31.522, Z 42.500}
   LaserEnd_Ext()
   LIN {X 4.428, Y 30.522, Z 42.500}
   LaserStart_Ext()
   LIN {X -2.456, Y 30.522, Z 42.500}
   LaserEnd_Ext()
   LIN {X -2.265, Y 29.522, Z 42.500}
   LaserStart_Ext()
   LIN {X 4.719, Y 29.522, Z 42.500}
   LaserEnd_Ext()
   LIN {X 4.980, Y 28.522, Z 42.500}
   LaserStart_Ext()
   LIN {X -2.074, Y 28.522, Z 42.500}
   LaserEnd_Ext()
   LIN {X -1.906, Y 27.522, Z 42.500}
   LaserStart_Ext()
   LIN {X 5.214, Y 27.522, Z 42.500}
   LaserEnd_Ext()
   LIN {X 5.448, Y 26.522, Z 42.500}
   LaserStart_Ext()
   LIN {X -1.778, Y 26.522, Z 42.500}
   LaserEnd_Ext()
   LIN {X -1.650, Y 25.522, Z 42.500}
   LaserStart_Ext()
   LIN {X 5.683, Y 25.522, Z 42.500}
   LaserEnd_Ext()
   LIN {X 5.918, Y 24.522, Z 42.500}
   LaserStart_Ext()
   LIN {X -1.522, Y 24.522, Z 42.500}
   LaserEnd_Ext()
   LIN {X -1.394, Y 23.522, Z 42.500}
   LaserStart_Ext()
   LIN {X 6.155, Y 23.522, Z 42.500}
   LaserEnd_Ext()
   LIN {X 6.386, Y 22.522, Z 42.500}
   LaserStart_Ext()
   LIN {X -1.277, Y 22.522, Z 42.500}
   LaserEnd_Ext()
   LIN {X -1.272, Y 21.522, Z 42.500}
   LaserStart_Ext()
   LIN {X 6.545, Y 21.522, Z 42.500}
   LaserEnd_Ext()
   LIN {X 6.696, Y 20.522, Z 42.500}
   LaserStart_Ext()
   LIN {X -1.267, Y 20.522, Z 42.500}
   LaserEnd_Ext()
   LIN {X -1.260, Y 19.522, Z 42.500}
   LaserStart_Ext()
   LIN {X 6.847, Y 19.522, Z 42.500}
   LaserEnd_Ext()
   LIN {X 6.998, Y 18.522, Z 42.500}
   LaserStart_Ext()
   LIN {X -1.219, Y 18.522, Z 42.500}
   LaserEnd_Ext()
   LIN {X -1.178, Y 17.522, Z 42.500}
   LaserStart_Ext()
   LIN {X 7.149, Y 17.522, Z 42.500}
   LaserEnd_Ext()
   LIN {X 7.300, Y 16.522, Z 42.500}
   LaserStart_Ext()
   LIN {X -1.137, Y 16.522, Z 42.500}
   LaserEnd_Ext()
   LIN {X -1.096, Y 15.522, Z 42.500}
   LaserStart_Ext()
   LIN {X 7.450, Y 15.522, Z 42.500}
   LaserEnd_Ext()
   LIN {X 7.601, Y 14.522, Z 42.500}
   LaserStart_Ext()
   LIN {X -1.055, Y 14.522, Z 42.500}
   LaserEnd_Ext()
   LIN {X -1.014, Y 13.522, Z 42.500}
   LaserStart_Ext()
   LIN {X 7.752, Y 13.522, Z 42.500}
   LaserEnd_Ext()
   LIN {X 7.863, Y 12.522, Z 42.500}
   LaserStart_Ext()
   LIN {X -0.984, Y 12.522, Z 42.500}
   LaserEnd_Ext()
   LIN {X -1.089, Y 11.522, Z 42.500}
   LaserStart_Ext()
   LIN {X 7.948, Y 11.522, Z 42.500}
   LaserEnd_Ext()
   LIN {X 8.033, Y 10.522, Z 42.500}
   LaserStart_Ext()
   LIN {X -1.195, Y 10.522, Z 42.500}
   LaserEnd_Ext()
   LIN {X -1.301, Y 9.522, Z 42.500}
   LaserStart_Ext()
   LIN {X 8.118, Y 9.522, Z 42.500}
   LaserEnd_Ext()
   LIN {X 8.204, Y 8.522, Z 42.500}
   LaserStart_Ext()
   LIN {X -1.407, Y 8.522, Z 42.500}
   LaserEnd_Ext()
   LIN {X -1.513, Y 7.522, Z 42.500}
   LaserStart_Ext()
   LIN {X 8.289, Y 7.522, Z 42.500}
   LaserEnd_Ext()
   LIN {X 8.374, Y 6.522, Z 42.500}
   LaserStart_Ext()
   LIN {X -1.619, Y 6.522, Z 42.500}
   LaserEnd_Ext()
   LIN {X -1.711, Y 5.522, Z 42.500}
   LaserStart_Ext()
   LIN {X 8.459, Y 5.522, Z 42.500}
   LaserEnd_Ext()
   LIN {X 8.507, Y 4.522, Z 42.500}
   LaserStart_Ext()
   LIN {X -1.790, Y 4.522, Z 42.500}
   LaserEnd_Ext()
   LIN {X -1.948, Y 3.522, Z 42.500}
   LaserStart_Ext()
   LIN {X 8.508, Y 3.522, Z 42.500}
   LaserEnd_Ext()
   LIN {X 8.508, Y 2.522, Z 42.500}
   LaserStart_Ext()
   LIN {X -2.145, Y 2.522, Z 42.500}
   LaserEnd_Ext()
   LIN {X -2.342, Y 1.522, Z 42.500}
   LaserStart_Ext()
   LIN {X 8.509, Y 1.522, Z 42.500}
   LaserEnd_Ext()
   LIN {X 8.510, Y 0.522, Z 42.500}
   LaserStart_Ext()
   LIN {X -2.539, Y 0.522, Z 42.500}
   LaserEnd_Ext()
   LIN {X -2.744, Y -0.478, Z 42.500}
   LaserStart_Ext()
   LIN {X 8.511, Y -0.478, Z 42.500}
   LaserEnd_Ext()
   LIN {X 8.512, Y -1.478, Z 42.500}
   LaserStart_Ext()
   LIN {X -2.955, Y -1.478, Z 42.500}
   LaserEnd_Ext()
   LIN {X -3.205, Y -2.478, Z 42.500}
   LaserStart_Ext()
   LIN {X 8.512, Y -2.478, Z 42.500}
   LaserEnd_Ext()
   LIN {X 8.503, Y -3.478, Z 42.500}
   LaserStart_Ext()
   LIN {X -3.487, Y -3.478, Z 42.500}
   LaserEnd_Ext()
   LIN {X -3.764, Y -4.478, Z 42.500}
   LaserStart_Ext()
   LIN {X 8.444, Y -4.478, Z 42.500}
   LaserEnd_Ext()
   LIN {X 8.384, Y -5.478, Z 42.500}
   LaserStart_Ext()
   LIN {X -4.038, Y -5.478, Z 42.500}
   LaserEnd_Ext()
   LIN {X -4.323, Y -6.478, Z 42.500}
   LaserStart_Ext()
   LIN {X 8.324, Y -6.478, Z 42.500}
   LaserEnd_Ext()
   LIN {X 8.258, Y -7.478, Z 42.500}
   LaserStart_Ext()
   LIN {X -4.668, Y -7.478, Z 42.500}
   LaserEnd_Ext()
   LIN {X -5.013, Y -8.478, Z 42.500}
   LaserStart_Ext()
   LIN {X 8.192, Y -8.478, Z 42.500}
   LaserEnd_Ext()
   LIN {X 8.097, Y -9.478, Z 42.500}
   LaserStart_Ext()
   LIN {X -5.363, Y -9.478, Z 42.500}
   LaserEnd_Ext()
   LIN {X -5.715, Y -10.478, Z 42.500}
   LaserStart_Ext()
   LIN {X 7.985, Y -10.478, Z 42.500}
   LaserEnd_Ext()
   LIN {X 7.874, Y -11.478, Z 42.500}
   LaserStart_Ext()
   LIN {X -6.106, Y -11.478, Z 42.500}
   LaserEnd_Ext()
   LIN {X -6.525, Y -12.478, Z 42.500}
   LaserStart_Ext()
   LIN {X 7.766, Y -12.478, Z 42.500}
   LaserEnd_Ext()
   LIN {X 7.660, Y -13.478, Z 42.500}
   LaserStart_Ext()
   LIN {X -6.940, Y -13.478, Z 42.500}
   LaserEnd_Ext()
   LIN {X -7.352, Y -14.478, Z 42.500}
   LaserStart_Ext()
   LIN {X 7.518, Y -14.478, Z 42.500}
   LaserEnd_Ext()
   LIN {X 7.368, Y -15.478, Z 42.500}
   LaserStart_Ext()
   LIN {X -7.825, Y -15.478, Z 42.500}
   LaserEnd_Ext()
   LIN {X -8.306, Y -16.478, Z 42.500}
   LaserStart_Ext()
   LIN {X -4.932, Y -16.478, Z 42.500}
   LaserEnd_Ext()
   LIN {X 1.066, Y -16.478, Z 42.500}
   LaserStart_Ext()
   LIN {X 7.217, Y -16.478, Z 42.500}
   LaserEnd_Ext()
   LIN {X 7.058, Y -17.478, Z 42.500}
   LaserStart_Ext()
   LIN {X 2.483, Y -17.478, Z 42.500}
   LaserEnd_Ext()
   LIN {X -6.098, Y -17.478, Z 42.500}
   LaserStart_Ext()
   LIN {X -8.787, Y -17.478, Z 42.500}
   LaserEnd_Ext()
   LIN {X -9.168, Y -18.478, Z 42.500}
   LaserStart_Ext()
   LIN {X -6.926, Y -18.478, Z 42.500}
   LaserEnd_Ext()
   LIN {X 3.059, Y -18.478, Z 42.500}
   LaserStart_Ext()
   LIN {X 6.876, Y -18.478, Z 42.500}
   LaserEnd_Ext()
   LIN {X 6.695, Y -19.478, Z 42.500}
   LaserStart_Ext()
   LIN {X 3.616, Y -19.478, Z 42.500}
   LaserEnd_Ext()
   LIN {X -7.297, Y -19.478, Z 42.500}
   LaserStart_Ext()
   LIN {X -9.474, Y -19.478, Z 42.500}
   LaserEnd_Ext()
   LIN {X -9.781, Y -20.478, Z 42.500}
   LaserStart_Ext()
   LIN {X -7.666, Y -20.478, Z 42.500}
   LaserEnd_Ext()
   LIN {X 3.953, Y -20.478, Z 42.500}
   LaserStart_Ext()
   LIN {X 6.509, Y -20.478, Z 42.500}
   LaserEnd_Ext()
   LIN {X 6.301, Y -21.478, Z 42.500}
   LaserStart_Ext()
   LIN {X 3.981, Y -21.478, Z 42.500}
   LaserEnd_Ext()
   LIN {X -7.882, Y -21.478, Z 42.500}
   LaserStart_Ext()
   LIN {X -9.772, Y -21.478, Z 42.500}
   LaserEnd_Ext()
   LIN {X -9.685, Y -22.478, Z 42.500}
   LaserStart_Ext()
   LIN {X -7.742, Y -22.478, Z 42.500}
   LaserEnd_Ext()
   LIN {X 4.009, Y -22.478, Z 42.500}
   LaserStart_Ext()
   LIN {X 6.091, Y -22.478, Z 42.500}
   LaserEnd_Ext()
   LIN {X 5.832, Y -23.478, Z 42.500}
   LaserStart_Ext()
   LIN {X 3.667, Y -23.478, Z 42.500}
   LaserEnd_Ext()
   LIN {X -7.599, Y -23.478, Z 42.500}
   LaserStart_Ext()
   LIN {X -9.599, Y -23.478, Z 42.500}
   LaserEnd_Ext()
   LIN {X -9.271, Y -24.478, Z 42.500}
   LaserStart_Ext()
   LIN {X -7.077, Y -24.478, Z 42.500}
   LaserEnd_Ext()
   LIN {X 3.209, Y -24.478, Z 42.500}
   LaserStart_Ext()
   LIN {X 5.426, Y -24.478, Z 42.500}
   LaserEnd_Ext()
   LIN {X 5.019, Y -25.478, Z 42.500}
   LaserStart_Ext()
   LIN {X 2.616, Y -25.478, Z 42.500}
   LaserEnd_Ext()
   LIN {X -6.440, Y -25.478, Z 42.500}
   LaserStart_Ext()
   LIN {X -8.716, Y -25.478, Z 42.500}
   LaserEnd_Ext()
   LIN {X -8.164, Y -26.478, Z 42.500}
   LaserStart_Ext()
   LIN {X -5.243, Y -26.478, Z 42.500}
   LaserEnd_Ext()
   LIN {X 1.399, Y -26.478, Z 42.500}
   LaserStart_Ext()
   LIN {X 4.247, Y -26.478, Z 42.500}
   LaserEnd_Ext()
   LIN {X 3.365, Y -27.478, Z 42.500}
   LaserStart_Ext()
   LIN {X -1.170, Y -27.478, Z 42.500}
   LaserEnd_Ext()
   LIN {X -2.531, Y -27.478, Z 42.500}
   LaserStart_Ext()
   LIN {X -7.233, Y -27.478, Z 42.500}
   LaserEnd_Ext()
   LIN {X -6.017, Y -28.478, Z 42.500}
   LaserStart_Ext()
   LIN {X 1.825, Y -28.478, Z 42.500}
   LaserEnd_Ext()
   LIN {X -2.131, Y -29.478, Z 42.500}
   LaserStart_Ext()
   LIN {X -3.004, Y -29.478, Z 42.500}
   LaserEnd_Ext()
   LIN {X -4.544, Y -17.485, Z 43.350}
   LaserStart_Ext()
   LIN {X -4.090, Y -17.097, Z 43.350} C_DIS
   LIN {X -3.443, Y -16.912, Z 43.350} C_DIS
   LIN {X -2.059, Y -16.551, Z 43.350} C_DIS
   LIN {X -0.940, Y -16.729, Z 43.350} C_DIS
   LIN {X 0.013, Y -16.878, Z 43.350} C_DIS
   LIN {X 1.024, Y -17.551, Z 43.350} C_DIS
   LIN {X 1.780, Y -18.057, Z 43.350} C_DIS
   LIN {X 2.264, Y -18.924, Z 43.350} C_DIS
   LIN {X 3.023, Y -20.276, Z 43.350} C_DIS
   LIN {X 3.061, Y -21.464, Z 43.350} C_DIS
   LIN {X 3.089, Y -22.451, Z 43.350} C_DIS
   LIN {X 2.795, Y -23.091, Z 43.350} C_DIS
   LIN {X 2.081, Y -24.643, Z 43.350} C_DIS
   LIN {X 0.412, Y -26.008, Z 43.350} C_DIS
   LIN {X -1.661, Y -26.545, Z 43.350} C_DIS
   LIN {X -3.061, Y -26.316, Z 43.350} C_DIS
   LIN {X -3.680, Y -26.212, Z 43.350} C_DIS
   LIN {X -4.368, Y -25.755, Z 43.350} C_DIS
   LIN {X -5.403, Y -25.073, Z 43.350} C_DIS
   LIN {X -5.932, Y -24.250, Z 43.350} C_DIS
   LIN {X -6.526, Y -23.319, Z 43.350} C_DIS
   LIN {X -6.690, Y -22.163, Z 43.350} C_DIS
   LIN {X -6.823, Y -21.253, Z 43.350} C_DIS
   LIN {X -6.388, Y -20.103, Z 43.350} C_DIS
   LIN {X -5.808, Y -18.539, Z 43.350} C_DIS
   LIN {X -4.544, Y -17.485, Z 43.350}
   LaserEnd_Ext()
   LIN {X 2.522, Y 39.457, Z 43.350}
   LaserStart_Ext()
   LIN {X 3.103, Y 37.890, Z 43.350} C_DIS
   LIN {X 3.743, Y 36.051, Z 43.350} C_DIS
   LIN {X 4.169, Y 34.749, Z 43.350} C_DIS
   LIN {X 4.272, Y 34.433, Z 43.350} C_DIS
   LIN {X 4.528, Y 33.656, Z 43.350} C_DIS
   LIN {X 5.770, Y 29.382, Z 43.350} C_DIS
   LIN {X 5.835, Y 29.153, Z 43.350} C_DIS
   LIN {X 7.201, Y 23.398, Z 43.350} C_DIS
   LIN {X 7.513, Y 21.908, Z 43.350} C_DIS
   LIN {X 8.742, Y 13.766, Z 43.350} C_DIS
   LIN {X 9.385, Y 6.217, Z 43.350} C_DIS
   LIN {X 9.531, Y 4.866, Z 43.350} C_DIS
   LIN {X 9.542, Y 2.968, Z 43.350} C_DIS
   LIN {X 9.547, Y -3.259, Z 43.350} C_DIS
   LIN {X 9.243, Y -8.381, Z 43.350} C_DIS
   LIN {X 9.212, Y -8.842, Z 43.350} C_DIS
   LIN {X 9.158, Y -9.333, Z 43.350} C_DIS
   LIN {X 8.705, Y -13.578, Z 43.350} C_DIS
   LIN {X 8.364, Y -15.947, Z 43.350} C_DIS
   LIN {X 8.153, Y -17.344, Z 43.350} C_DIS
   LIN {X 7.937, Y -18.531, Z 43.350} C_DIS
   LIN {X 7.634, Y -20.259, Z 43.350} C_DIS
   LIN {X 7.247, Y -22.157, Z 43.350} C_DIS
   LIN {X 6.974, Y -23.454, Z 43.350} C_DIS
   LIN {X 6.250, Y -25.237, Z 43.350} C_DIS
   LIN {X 5.843, Y -26.229, Z 43.350} C_DIS
   LIN {X 5.444, Y -26.678, Z 43.350} C_DIS
   LIN {X 3.780, Y -28.566, Z 43.350} C_DIS
   LIN {X 1.517, Y -29.775, Z 43.350} C_DIS
   LIN {X 0.731, Y -30.168, Z 43.350} C_DIS
   LIN {X -0.233, Y -30.249, Z 43.350} C_DIS
   LIN {X -2.929, Y -30.496, Z 43.350} C_DIS
   LIN {X -4.887, Y -29.844, Z 43.350} C_DIS
   LIN {X -6.385, Y -29.354, Z 43.350} C_DIS
   LIN {X -8.170, Y -27.886, Z 43.350} C_DIS
   LIN {X -8.631, Y -27.509, Z 43.350} C_DIS
   LIN {X -8.813, Y -27.186, Z 43.350} C_DIS
   LIN {X -10.453, Y -24.232, Z 43.350} C_DIS
   LIN {X -10.678, Y -21.623, Z 43.350} C_DIS
   LIN {X -10.780, Y -20.536, Z 43.350} C_DIS
   LIN {X -10.325, Y -19.029, Z 43.350} C_DIS
   LIN {X -9.856, Y -17.503, Z 43.350} C_DIS
   LIN {X -9.283, Y -16.311, Z 43.350} C_DIS
   LIN {X -8.204, Y -14.030, Z 43.350} C_DIS
   LIN {X -6.983, Y -11.063, Z 43.350} C_DIS
   LIN {X -6.732, Y -10.463, Z 43.350} C_DIS
   LIN {X -6.530, Y -9.890, Z 43.350} C_DIS
   LIN {X -5.206, Y -6.054, Z 43.350} C_DIS
   LIN {X -4.160, Y -2.235, Z 43.350} C_DIS
   LIN {X -3.974, Y -1.579, Z 43.350} C_DIS
   LIN {X -3.827, Y -0.880, Z 43.350} C_DIS
   LIN {X -2.798, Y 4.340, Z 43.350} C_DIS
   LIN {X -2.613, Y 6.681, Z 43.350} C_DIS
   LIN {X -1.983, Y 12.627, Z 43.350} C_DIS
   LIN {X -2.311, Y 20.646, Z 43.350} C_DIS
   LIN {X -2.323, Y 22.814, Z 43.350} C_DIS
   LIN {X -2.799, Y 26.530, Z 43.350} C_DIS
   LIN {X -3.001, Y 27.890, Z 43.350} C_DIS
   LIN {X -3.167, Y 28.695, Z 43.350} C_DIS
   LIN {X -3.267, Y 29.227, Z 43.350} C_DIS
   LIN {X -3.601, Y 30.988, Z 43.350} C_DIS
   LIN {X -3.874, Y 32.131, Z 43.350} C_DIS
   LIN {X -4.259, Y 33.759, Z 43.350} C_DIS
   LIN {X -4.492, Y 34.612, Z 43.350} C_DIS
   LIN {X -4.888, Y 36.045, Z 43.350} C_DIS
   LIN {X -5.327, Y 37.482, Z 43.350} C_DIS
   LIN {X -5.370, Y 37.622, Z 43.350} C_DIS
   LIN {X -5.738, Y 38.767, Z 43.350} C_DIS
   LIN {X -5.927, Y 39.990, Z 43.350} C_DIS
   LIN {X -5.951, Y 40.150, Z 43.350} C_DIS
   LIN {X -5.889, Y 40.391, Z 43.350} C_DIS
   LIN {X -5.524, Y 41.842, Z 43.350} C_DIS
   LIN {X -4.993, Y 42.516, Z 43.350} C_DIS
   LIN {X -4.557, Y 43.070, Z 43.350} C_DIS
   LIN {X -2.190, Y 44.013, Z 43.350} C_DIS
   LIN {X -1.551, Y 43.905, Z 43.350} C_DIS
   LIN {X -0.469, Y 43.720, Z 43.350} C_DIS
   LIN {X 0.894, Y 42.773, Z 43.350} C_DIS
   LIN {X 0.990, Y 42.681, Z 43.350} C_DIS
   LIN {X 1.746, Y 41.480, Z 43.350} C_DIS
   LIN {X 2.189, Y 40.344, Z 43.350} C_DIS
   LIN {X 2.286, Y 40.096, Z 43.350} C_DIS
   LIN {X 2.522, Y 39.457, Z 43.350}
   LaserEnd_Ext()
   LIN {X -9.280, Y -24.284, Z 43.350}
   LaserStart_Ext()
   LIN {X -9.280, Y -19.032, Z 43.350}
   LaserEnd_Ext()
   LIN {X -8.280, Y -16.530, Z 43.350}
   LaserStart_Ext()
   LIN {X -8.280, Y -26.086, Z 43.350}
   LaserEnd_Ext()
   LIN {X -7.280, Y -27.323, Z 43.350}
   LaserStart_Ext()
   LIN {X -7.280, Y -23.996, Z 43.350}
   LaserEnd_Ext()
   LIN {X -7.280, Y -19.631, Z 43.350}
   LaserStart_Ext()
   LIN {X -7.280, Y -14.413, Z 43.350}
   LaserEnd_Ext()
   LIN {X -6.280, Y -11.983, Z 43.350}
   LaserStart_Ext()
   LIN {X -6.280, Y -17.631, Z 43.350}
   LaserEnd_Ext()
   LIN {X -6.280, Y -25.558, Z 43.350}
   LaserStart_Ext()
   LIN {X -6.280, Y -28.146, Z 43.350}
   LaserEnd_Ext()
   LIN {X -5.280, Y -28.663, Z 43.350}
   LaserStart_Ext()
   LIN {X -5.280, Y -26.352, Z 43.350}
   LaserEnd_Ext()
   LIN {X -5.280, Y -16.796, Z 43.350}
   LaserStart_Ext()
   LIN {X -5.280, Y -9.334, Z 43.350}
   LaserEnd_Ext()
   LIN {X -4.280, Y 41.805, Z 43.350}
   LaserStart_Ext()
   LIN {X -4.280, Y 37.478, Z 43.350}
   LaserEnd_Ext()
   LIN {X -4.280, Y -6.437, Z 43.350}
   LaserStart_Ext()
   LIN {X -4.280, Y -16.111, Z 43.350}
   LaserEnd_Ext()
   LIN {X -4.280, Y -27.015, Z 43.350}
   LaserStart_Ext()
   LIN {X -4.280, Y -28.992, Z 43.350}
   LaserEnd_Ext()
   LIN {X -3.280, Y -29.325, Z 43.350}
   LaserStart_Ext()
   LIN {X -3.280, Y -27.293, Z 43.350}
   LaserEnd_Ext()
   LIN {X -3.280, Y -15.836, Z 43.350}
   LaserStart_Ext()
   LIN {X -3.280, Y -2.809, Z 43.350}
   LaserEnd_Ext()
   LIN {X -3.280, Y 33.965, Z 43.350}
   LaserStart_Ext()
   LIN {X -3.280, Y 42.502, Z 43.350}
   LaserEnd_Ext()
   LIN {X -2.280, Y 42.901, Z 43.350}
   LaserStart_Ext()
   LIN {X -2.280, Y 29.386, Z 43.350}
   LaserEnd_Ext()
   LIN {X -2.280, Y 1.798, Z 43.350}
   LaserStart_Ext()
   LIN {X -2.280, Y -15.577, Z 43.350}
   LaserEnd_Ext()
   LIN {X -2.280, Y -27.457, Z 43.350}
   LaserStart_Ext()
   LIN {X -2.280, Y -29.433, Z 43.350}
   LaserEnd_Ext()
   LIN {X -1.280, Y -29.341, Z 43.350}
   LaserStart_Ext()
   LIN {X -1.280, Y -27.480, Z 43.350}
   LaserEnd_Ext()
   LIN {X -1.280, Y -15.662, Z 43.350}
   LaserStart_Ext()
   LIN {X -1.280, Y 9.770, Z 43.350}
   LaserEnd_Ext()
   LIN {X -1.280, Y 19.894, Z 43.350}
   LaserStart_Ext()
   LIN {X -1.280, Y 42.844, Z 43.350}
   LaserEnd_Ext()
   LIN {X -0.280, Y 42.371, Z 43.350}
   LaserStart_Ext()
   LIN {X -0.280, Y -15.820, Z 43.350}
   LaserEnd_Ext()
   LIN {X -0.280, Y -27.221, Z 43.350}
   LaserStart_Ext()
   LIN {X -0.280, Y -29.250, Z 43.350}
   LaserEnd_Ext()
   LIN {X 0.720, Y -29.056, Z 43.350}
   LaserStart_Ext()
   LIN {X 0.720, Y -26.960, Z 43.350}
   LaserEnd_Ext()
   LIN {X 0.720, Y -16.147, Z 43.350}
   LaserStart_Ext()
   LIN {X 0.720, Y 41.232, Z 43.350}
   LaserEnd_Ext()
   LIN {X 1.720, Y 38.742, Z 43.350}
   LaserStart_Ext()
   LIN {X 1.720, Y -16.813, Z 43.350}
   LaserEnd_Ext()
   LIN {X 1.720, Y -26.230, Z 43.350}
   LaserStart_Ext()
   LIN {X 1.720, Y -28.533, Z 43.350}
   LaserEnd_Ext()
   LIN {X 2.720, Y -27.998, Z 43.350}
   LaserStart_Ext()
   LIN {X 2.720, Y -25.412, Z 43.350}
   LaserEnd_Ext()
   LIN {X 2.720, Y -17.689, Z 43.350}
   LaserStart_Ext()
   LIN {X 2.720, Y 35.948, Z 43.350}
   LaserEnd_Ext()
   LIN {X 3.720, Y 32.851, Z 43.350}
   LaserStart_Ext()
   LIN {X 3.720, Y -19.475, Z 43.350}
   LaserEnd_Ext()
   LIN {X 3.720, Y -23.474, Z 43.350}
   LaserStart_Ext()
   LIN {X 3.720, Y -27.122, Z 43.350}
   LaserEnd_Ext()
   LIN {X 4.720, Y -25.988, Z 43.350}
   LaserStart_Ext()
   LIN {X 4.720, Y 29.410, Z 43.350}
   LaserEnd_Ext()
   LIN {X 5.720, Y 25.308, Z 43.350}
   LaserStart_Ext()
   LIN {X 5.720, Y -23.884, Z 43.350}
   LaserEnd_Ext()
   LIN {X 6.720, Y -19.680, Z 43.350}
   LaserStart_Ext()
   LIN {X 6.720, Y 20.461, Z 43.350}
   LaserEnd_Ext()
   LIN {X 7.720, Y 13.835, Z 43.350}
   LaserStart_Ext()
   LIN {X 7.720, Y -13.383, Z 43.350}
   LaserEnd_Ext()
   LIN {X -4.140, Y -25.809, Z 44.200}
   LaserStart_Ext()
   LIN {X -5.318, Y -25.032, Z 44.200} C_DIS
   LIN {X -6.286, Y -23.526, Z 44.200} C_DIS
   LIN {X -6.445, Y -23.280, Z 44.200} C_DIS
   LIN {X -6.490, Y -22.980, Z 44.200} C_DIS
   LIN {X -6.747, Y -21.215, Z 44.200} C_DIS
   LIN {X -5.793, Y -18.690, Z 44.200} C_DIS
   LIN {X -5.709, Y -18.461, Z 44.200} C_DIS
   LIN {X -5.622, Y -18.380, Z 44.200} C_DIS
   LIN {X -4.152, Y -17.125, Z 44.200} C_DIS
   LIN {X -2.202, Y -16.569, Z 44.200} C_DIS
   LIN {X -1.988, Y -16.502, Z 44.200} C_DIS
   LIN {X 0.079, Y -16.824, Z 44.200} C_DIS
   LIN {X 1.333, Y -17.659, Z 44.200} C_DIS
   LIN {X 1.849, Y -17.999, Z 44.200} C_DIS
   LIN {X 2.245, Y -18.699, Z 44.200} C_DIS
   LIN {X 3.097, Y -20.215, Z 44.200} C_DIS
   LIN {X 3.150, Y -21.890, Z 44.200} C_DIS
   LIN {X 3.168, Y -22.390, Z 44.200} C_DIS
   LIN {X 3.075, Y -22.613, Z 44.200} C_DIS
   LIN {X 2.171, Y -24.576, Z 44.200} C_DIS
   LIN {X 1.897, Y -24.816, Z 44.200} C_DIS
   LIN {X 0.539, Y -25.934, Z 44.200} C_DIS
   LIN {X -0.734, Y -26.279, Z 44.200} C_DIS
   LIN {X -1.573, Y -26.495, Z 44.200} C_DIS
   LIN {X -2.721, Y -26.307, Z 44.200} C_DIS
   LIN {X -3.592, Y -26.167, Z 44.200} C_DIS
   LIN {X -4.140, Y -25.809, Z 44.200}
   LaserEnd_Ext()
   LIN {X -5.802, Y 38.807, Z 44.200}
   LaserStart_Ext()
   LIN {X -5.738, Y 38.611, Z 44.200} C_DIS
   LIN {X -5.417, Y 37.616, Z 44.200} C_DIS
   LIN {X -5.073, Y 36.503, Z 44.200} C_DIS
   LIN {X -4.946, Y 36.087, Z 44.200} C_DIS
   LIN {X -4.703, Y 35.208, Z 44.200} C_DIS
   LIN {X -4.311, Y 33.802, Z 44.200} C_DIS
   LIN {X -3.959, Y 32.347, Z 44.200} C_DIS
   LIN {X -3.680, Y 31.179, Z 44.200} C_DIS
   LIN {X -3.579, Y 30.648, Z 44.200} C_DIS
   LIN {X -3.383, Y 29.607, Z 44.200} C_DIS
   LIN {X -3.057, Y 28.032, Z 44.200} C_DIS
   LIN {X -2.662, Y 25.371, Z 44.200} C_DIS
   LIN {X -2.368, Y 23.077, Z 44.200} C_DIS
   LIN {X -2.361, Y 21.739, Z 44.200} C_DIS
   LIN {X -1.988, Y 12.630, Z 44.200} C_DIS
   LIN {X -2.560, Y 7.226, Z 44.200} C_DIS
   LIN {X -2.788, Y 4.354, Z 44.200} C_DIS
   LIN {X -3.566, Y 0.403, Z 44.200} C_DIS
   LIN {X -3.939, Y -1.517, Z 44.200} C_DIS
   LIN {X -4.128, Y -2.216, Z 44.200} C_DIS
   LIN {X -5.187, Y -6.084, Z 44.200} C_DIS
   LIN {X -6.408, Y -9.619, Z 44.200} C_DIS
   LIN {X -6.695, Y -10.465, Z 44.200} C_DIS
   LIN {X -6.984, Y -11.175, Z 44.200} C_DIS
   LIN {X -8.145, Y -13.996, Z 44.200} C_DIS
   LIN {X -9.784, Y -17.460, Z 44.200} C_DIS
   LIN {X -10.705, Y -20.507, Z 44.200} C_DIS
   LIN {X -10.499, Y -22.705, Z 44.200} C_DIS
   LIN {X -10.370, Y -24.203, Z 44.200} C_DIS
   LIN {X -9.429, Y -25.899, Z 44.200} C_DIS
   LIN {X -8.540, Y -27.475, Z 44.200} C_DIS
   LIN {X -6.291, Y -29.315, Z 44.200} C_DIS
   LIN {X -5.802, Y 38.807, Z 44.200}
   LaserEnd_Ext()
   LIN {X 7.055, Y -23.384, Z 44.200}
   LaserStart_Ext()
   LIN {X 6.992, Y -23.540, Z 44.200} C_DIS
   LIN {X 5.889, Y -26.228, Z 44.200} C_DIS
   LIN {X 4.808, Y -27.446, Z 44.200} C_DIS
   LIN {X 3.882, Y -28.496, Z 44.200} C_DIS
   LIN {X 1.676, Y -29.675, Z 44.200} C_DIS
   LIN {X 0.911, Y -30.090, Z 44.200} C_DIS
   LIN {X 0.543, Y -30.120, Z 44.200} C_DIS
   LIN {X -2.922, Y -30.438, Z 44.200} C_DIS
   LIN {X -6.289, Y -29.316, Z 44.200} C_DIS
   LIN {X 7.055, Y -23.384, Z 44.200}
   LaserEnd_Ext()
   LIN {X 1.675, Y 41.538, Z 44.200}
   LaserStart_Ext()
   LIN {X 1.629, Y 41.610, Z 44.200} C_DIS
   LIN {X 0.888, Y 42.782, Z 44.200} C_DIS
   LIN {X -0.316, Y 43.615, Z 44.200} C_DIS
   LIN {X -0.545, Y 43.772, Z 44.200} C_DIS
   LIN {X -1.014, Y 43.850, Z 44.200} C_DIS
   LIN {X -2.267, Y 44.061, Z 44.200} C_DIS
   LIN {X -4.616, Y 43.125, Z 44.200} C_DIS
   LIN {X -5.247, Y 42.324, Z 44.200} C_DIS
   LIN {X -5.582, Y 41.908, Z 44.200} C_DIS
   LIN {X -5.756, Y 41.267, Z 44.200} C_DIS
   LIN {X -6.017, Y 40.240, Z 44.200} C_DIS
   LIN {X -5.855, Y 39.168, Z 44.200} C_DIS
   LIN {X 1.675, Y 41.538, Z 44.200}
   LaserEnd_Ext()
   LIN {X 7.055, Y -23.384, Z 44.200}
   LaserStart_Ext()
   LIN {X 7.079, Y -23.271, Z 44.200} C_DIS
   LIN {X 7.708, Y -20.187, Z 44.200} C_DIS
   LIN {X 8.200, Y -17.380, Z 44.200} C_DIS
   LIN {X 8.220, Y -17.271, Z 44.200} C_DIS
   LIN {X 8.239, Y -17.143, Z 44.200} C_DIS
   LIN {X 8.763, Y -13.504, Z 44.200} C_DIS
   LIN {X 9.142, Y -9.949, Z 44.200} C_DIS
   LIN {X 9.260, Y -8.760, Z 44.200} C_DIS
   LIN {X 9.359, Y -6.912, Z 44.200} C_DIS
   LIN {X 9.581, Y -3.178, Z 44.200} C_DIS
   LIN {X 9.578, Y 0.638, Z 44.200} C_DIS
   LIN {X 9.554, Y 4.819, Z 44.200} C_DIS
   LIN {X 9.232, Y 7.796, Z 44.200} C_DIS
   LIN {X 8.680, Y 14.276, Z 44.200} C_DIS
   LIN {X 7.625, Y 21.264, Z 44.200} C_DIS
   LIN {X 7.096, Y 23.796, Z 44.200} C_DIS
   LIN {X 5.919, Y 28.751, Z 44.200} C_DIS
   LIN {X 5.540, Y 30.082, Z 44.200} C_DIS
   LIN {X 4.560, Y 33.451, Z 44.200} C_DIS
   LIN {X 4.147, Y 34.710, Z 44.200} C_DIS
   LIN {X 3.979, Y 35.223, Z 44.200} C_DIS
   LIN {X 3.745, Y 35.942, Z 44.200} C_DIS
   LIN {X 3.260, Y 37.320, Z 44.200} C_DIS
   LIN {X 3.042, Y 37.946, Z 44.200} C_DIS
   LIN {X 2.718, Y 38.820, Z 44.200} C_DIS
   LIN {X 2.219, Y 40.152, Z 44.200} C_DIS
   LIN {X 1.715, Y 41.434, Z 44.200} C_DIS
   LIN {X 7.055, Y -23.384, Z 44.200}
   LaserEnd_Ext()
   LIN {X 2.015, Y -28.360, Z 44.200}
   LaserStart_Ext()
   LIN {X 1.749, Y -28.360, Z 44.200}
   LaserEnd_Ext()
   LIN {X 3.164, Y -27.360, Z 44.200}
   LaserStart_Ext()
   LIN {X 3.551, Y -27.360, Z 44.200}
   LaserEnd_Ext()
   LIN {X -2.318, Y -25.360, Z 44.200}
   LaserStart_Ext()
   LIN {X -1.176, Y -25.360, Z 44.200}
   LaserEnd_Ext()
   LIN {X 0.877, Y -24.360, Z 44.200}
   LaserStart_Ext()
   LIN {X -4.520, Y -24.360, Z 44.200}
   LaserEnd_Ext()
   LIN {X -5.204, Y -23.360, Z 44.200}
   LaserStart_Ext()
   LIN {X 1.630, Y -23.360, Z 44.200}
   LaserEnd_Ext()
   LIN {X 2.091, Y -22.360, Z 44.200}
   LaserStart_Ext()
   LIN {X -5.569, Y -22.360, Z 44.200}
   LaserEnd_Ext()
   LIN {X -5.715, Y -21.360, Z 44.200}
   LaserStart_Ext()
   LIN {X 2.133, Y -21.360, Z 44.200}
   LaserEnd_Ext()
   LIN {X 2.031, Y -20.360, Z 44.200}
   LaserStart_Ext()
   LIN {X -5.355, Y -20.360, Z 44.200}
   LaserEnd_Ext()
   LIN {X -4.977, Y -19.360, Z 44.200}
   LaserStart_Ext()
   LIN {X 1.470, Y -19.360, Z 44.200}
   LaserEnd_Ext()
   LIN {X 0.583, Y -18.360, Z 44.200}
   LaserStart_Ext()
   LIN {X -4.058, Y -18.360, Z 44.200}
   LaserEnd_Ext()
   LIN {X 7.397, Y -15.360, Z 44.200}
   LaserStart_Ext()
   LIN {X 7.486, Y -15.360, Z 44.200}
   LaserEnd_Ext()
   LIN {X 7.630, Y -14.360, Z 44.200}
   LaserStart_Ext()
   LIN {X 7.315, Y -14.360, Z 44.200}
   LaserEnd_Ext()
   LIN {X 7.233, Y -13.360, Z 44.200}
   LaserStart_Ext()
   LIN {X 7.773, Y -13.360, Z 44.200}
   LaserEnd_Ext()
   LIN {X 7.879, Y -12.360, Z 44.200}
   LaserStart_Ext()
   LIN {X 7.150, Y -12.360, Z 44.200}
   LaserEnd_Ext()
   LIN {X 7.068, Y -11.360, Z 44.200}
   LaserStart_Ext()
   LIN {X 7.986, Y -11.360, Z 44.200}
   LaserEnd_Ext()
   LIN {X 8.093, Y -10.360, Z 44.200}
   LaserStart_Ext()
   LIN {X 6.986, Y -10.360, Z 44.200}
   LaserEnd_Ext()
   LIN {X 6.903, Y -9.360, Z 44.200}
   LaserStart_Ext()
   LIN {X 8.196, Y -9.360, Z 44.200}
   LaserEnd_Ext()
   LIN {X 8.280, Y -8.360, Z 44.200}
   LaserStart_Ext()
   LIN {X 6.821, Y -8.360, Z 44.200}
   LaserEnd_Ext()
   LIN {X -6.708, Y -7.360, Z 44.200}
   LaserStart_Ext()
   LIN {X -6.686, Y -7.360, Z 44.200}
   LaserEnd_Ext()
   LIN {X 6.738, Y -7.360, Z 44.200}
   LaserStart_Ext()
   LIN {X 8.334, Y -7.360, Z 44.200}
   LaserEnd_Ext()
   LIN {X 8.390, Y -6.360, Z 44.200}
   LaserStart_Ext()
   LIN {X 6.656, Y -6.360, Z 44.200}
   LaserEnd_Ext()
   LIN {X -6.341, Y -6.360, Z 44.200}
   LaserStart_Ext()
   LIN {X -6.667, Y -6.360, Z 44.200}
   LaserEnd_Ext()
   LIN {X -6.626, Y -5.360, Z 44.200}
   LaserStart_Ext()
   LIN {X -6.026, Y -5.360, Z 44.200}
   LaserEnd_Ext()
   LIN {X 6.574, Y -5.360, Z 44.200}
   LaserStart_Ext()
   LIN {X 8.450, Y -5.360, Z 44.200}
   LaserEnd_Ext()
   LIN {X 8.509, Y -4.360, Z 44.200}
   LaserStart_Ext()
   LIN {X 6.491, Y -4.360, Z 44.200}
   LaserEnd_Ext()
   LIN {X -5.752, Y -4.360, Z 44.200}
   LaserStart_Ext()
   LIN {X -6.585, Y -4.360, Z 44.200}
   LaserEnd_Ext()
   LIN {X -6.543, Y -3.360, Z 44.200}
   LaserStart_Ext()
   LIN {X -5.478, Y -3.360, Z 44.200}
   LaserEnd_Ext()
   LIN {X 6.409, Y -3.360, Z 44.200}
   LaserStart_Ext()
   LIN {X 8.568, Y -3.360, Z 44.200}
   LaserEnd_Ext()
   LIN {X 8.580, Y -2.360, Z 44.200}
   LaserStart_Ext()
   LIN {X 6.327, Y -2.360, Z 44.200}
   LaserEnd_Ext()
   LIN {X -5.204, Y -2.360, Z 44.200}
   LaserStart_Ext()
   LIN {X -6.502, Y -2.360, Z 44.200}
   LaserEnd_Ext()
   LIN {X -6.461, Y -1.360, Z 44.200}
   LaserStart_Ext()
   LIN {X -4.933, Y -1.360, Z 44.200}
   LaserEnd_Ext()
   LIN {X 6.244, Y -1.360, Z 44.200}
   LaserStart_Ext()
   LIN {X 8.580, Y -1.360, Z 44.200}
   LaserEnd_Ext()
   LIN {X 8.579, Y -0.360, Z 44.200}
   LaserStart_Ext()
   LIN {X 6.162, Y -0.360, Z 44.200}
   LaserEnd_Ext()
   LIN {X -4.733, Y -0.360, Z 44.200}
   LaserStart_Ext()
   LIN {X -6.419, Y -0.360, Z 44.200}
   LaserEnd_Ext()
   LIN {X -6.378, Y 0.640, Z 44.200}
   LaserStart_Ext()
   LIN {X -4.539, Y 0.640, Z 44.200}
   LaserEnd_Ext()
   LIN {X 6.079, Y 0.640, Z 44.200}
   LaserStart_Ext()
   LIN {X 8.578, Y 0.640, Z 44.200}
   LaserEnd_Ext()
   LIN {X 8.572, Y 1.640, Z 44.200}
   LaserStart_Ext()
   LIN {X 5.997, Y 1.640, Z 44.200}
   LaserEnd_Ext()
   LIN {X -4.342, Y 1.640, Z 44.200}
   LaserStart_Ext()
   LIN {X -6.337, Y 1.640, Z 44.200}
   LaserEnd_Ext()
   LIN {X -6.295, Y 2.640, Z 44.200}
   LaserStart_Ext()
   LIN {X -4.145, Y 2.640, Z 44.200}
   LaserEnd_Ext()
   LIN {X 5.915, Y 2.640, Z 44.200}
   LaserStart_Ext()
   LIN {X 8.566, Y 2.640, Z 44.200}
   LaserEnd_Ext()
   LIN {X 8.561, Y 3.640, Z 44.200}
   LaserStart_Ext()
   LIN {X 5.832, Y 3.640, Z 44.200}
   LaserEnd_Ext()
   LIN {X -3.948, Y 3.640, Z 44.200}
   LaserStart_Ext()
   LIN {X -6.254, Y 3.640, Z 44.200}
   LaserEnd_Ext()
   LIN {X -6.213, Y 4.640, Z 44.200}
   LaserStart_Ext()
   LIN {X -3.768, Y 4.640, Z 44.200}
   LaserEnd_Ext()
   LIN {X 5.750, Y 4.640, Z 44.200}
   LaserStart_Ext()
   LIN {X 8.555, Y 4.640, Z 44.200}
   LaserEnd_Ext()
   LIN {X 8.459, Y 5.640, Z 44.200}
   LaserStart_Ext()
   LIN {X 5.668, Y 5.640, Z 44.200}
   LaserEnd_Ext()
   LIN {X -3.689, Y 5.640, Z 44.200}
   LaserStart_Ext()
   LIN {X -6.172, Y 5.640, Z 44.200}
   LaserEnd_Ext()
   LIN {X -6.130, Y 6.640, Z 44.200}
   LaserStart_Ext()
   LIN {X -3.610, Y 6.640, Z 44.200}
   LaserEnd_Ext()
   LIN {X 5.585, Y 6.640, Z 44.200}
   LaserStart_Ext()
   LIN {X 8.351, Y 6.640, Z 44.200}
   LaserEnd_Ext()
   LIN {X 8.243, Y 7.640, Z 44.200}
   LaserStart_Ext()
   LIN {X 5.503, Y 7.640, Z 44.200}
   LaserEnd_Ext()
   LIN {X -3.522, Y 7.640, Z 44.200}
   LaserStart_Ext()
   LIN {X -6.089, Y 7.640, Z 44.200}
   LaserEnd_Ext()
   LIN {X -6.048, Y 8.640, Z 44.200}
   LaserStart_Ext()
   LIN {X -3.416, Y 8.640, Z 44.200}
   LaserEnd_Ext()
   LIN {X 5.420, Y 8.640, Z 44.200}
   LaserStart_Ext()
   LIN {X 8.157, Y 8.640, Z 44.200}
   LaserEnd_Ext()
   LIN {X 8.071, Y 9.640, Z 44.200}
   LaserStart_Ext()
   LIN {X 5.338, Y 9.640, Z 44.200}
   LaserEnd_Ext()
   LIN {X -3.310, Y 9.640, Z 44.200}
   LaserStart_Ext()
   LIN {X -6.006, Y 9.640, Z 44.200}
   LaserEnd_Ext()
   LIN {X -5.965, Y 10.640, Z 44.200}
   LaserStart_Ext()
   LIN {X -3.204, Y 10.640, Z 44.200}
   LaserEnd_Ext()
   LIN {X 5.256, Y 10.640, Z 44.200}
   LaserStart_Ext()
   LIN {X 7.986, Y 10.640, Z 44.200}
   LaserEnd_Ext()
   LIN {X 7.901, Y 11.640, Z 44.200}
   LaserStart_Ext()
   LIN {X 5.173, Y 11.640, Z 44.200}
   LaserEnd_Ext()
   LIN {X -3.098, Y 11.640, Z 44.200}
   LaserStart_Ext()
   LIN {X -5.924, Y 11.640, Z 44.200}
   LaserEnd_Ext()
   LIN {X -5.882, Y 12.640, Z 44.200}
   LaserStart_Ext()
   LIN {X -2.992, Y 12.640, Z 44.200}
   LaserEnd_Ext()
   LIN {X 5.091, Y 12.640, Z 44.200}
   LaserStart_Ext()
   LIN {X 7.816, Y 12.640, Z 44.200}
   LaserEnd_Ext()
   LIN {X 7.731, Y 13.640, Z 44.200}
   LaserStart_Ext()
   LIN {X 5.008, Y 13.640, Z 44.200}
   LaserEnd_Ext()
   LIN {X -3.030, Y 13.640, Z 44.200}
   LaserStart_Ext()
   LIN {X -5.841, Y 13.640, Z 44.200}
   LaserEnd_Ext()
   LIN {X -5.800, Y 14.640, Z 44.200}
   LaserStart_Ext()
   LIN {X -3.071, Y 14.640, Z 44.200}
   LaserEnd_Ext()
   LIN {X 4.926, Y 14.640, Z 44.200}
   LaserStart_Ext()
   LIN {X 7.614, Y 14.640, Z 44.200}
   LaserEnd_Ext()
   LIN {X 7.463, Y 15.640, Z 44.200}
   LaserStart_Ext()
   LIN {X 4.844, Y 15.640, Z 44.200}
   LaserEnd_Ext()
   LIN {X -3.112, Y 15.640, Z 44.200}
   LaserStart_Ext()
   LIN {X -5.758, Y 15.640, Z 44.200}
   LaserEnd_Ext()
   LIN {X -5.717, Y 16.640, Z 44.200}
   LaserStart_Ext()
   LIN {X -3.153, Y 16.640, Z 44.200}
   LaserEnd_Ext()
   LIN {X 4.761, Y 16.640, Z 44.200}
   LaserStart_Ext()
   LIN {X 7.312, Y 16.640, Z 44.200}
   LaserEnd_Ext()
   LIN {X 7.161, Y 17.640, Z 44.200}
   LaserStart_Ext()
   LIN {X 4.679, Y 17.640, Z 44.200}
   LaserEnd_Ext()
   LIN {X -3.194, Y 17.640, Z 44.200}
   LaserStart_Ext()
   LIN {X -5.676, Y 17.640, Z 44.200}
   LaserEnd_Ext()
   LIN {X -5.635, Y 18.640, Z 44.200}
   LaserStart_Ext()
   LIN {X -3.235, Y 18.640, Z 44.200}
   LaserEnd_Ext()
   LIN {X 4.597, Y 18.640, Z 44.200}
   LaserStart_Ext()
   LIN {X 7.010, Y 18.640, Z 44.200}
   LaserEnd_Ext()
   LIN {X 6.859, Y 19.640, Z 44.200}
   LaserStart_Ext()
   LIN {X 4.514, Y 19.640, Z 44.200}
   LaserEnd_Ext()
   LIN {X -3.276, Y 19.640, Z 44.200}
   LaserStart_Ext()
   LIN {X -5.593, Y 19.640, Z 44.200}
   LaserEnd_Ext()
   LIN {X -5.552, Y 20.640, Z 44.200}
   LaserStart_Ext()
   LIN {X -3.317, Y 20.640, Z 44.200}
   LaserEnd_Ext()
   LIN {X 4.432, Y 20.640, Z 44.200}
   LaserStart_Ext()
   LIN {X 6.708, Y 20.640, Z 44.200}
   LaserEnd_Ext()
   LIN {X 6.525, Y 21.640, Z 44.200}
   LaserStart_Ext()
   LIN {X 4.349, Y 21.640, Z 44.200}
   LaserEnd_Ext()
   LIN {X -3.358, Y 21.640, Z 44.200}
   LaserStart_Ext()
   LIN {X -5.511, Y 21.640, Z 44.200}
   LaserEnd_Ext()
   LIN {X -5.469, Y 22.640, Z 44.200}
   LaserStart_Ext()
